LIN {X 0,Y 473.146,Z 970.34,A -85,B 0,C 180,E1 12740.095,E2 12740.095} C_VEL
LIN {X 0,Y 467.036,Z 990.213,A -85,B 0,C 180,E1 12738.717,E2 12738.717} C_VEL
LIN {X 0,Y 459.248,Z 1013.166,A -85,B 0,C 180,E1 12736.833,E2 12736.833} C_VEL
LIN {X 0,Y 452.835,Z 1030.812,A -85,B 0,C 180,E1 12735.136,E2 12735.136} C_VEL
LIN {X 0,Y 446.449,Z 1047.58,A -85,B 0,C 180,E1 12733.29,E2 12733.29} C_VEL
LIN {X 0,Y 438.433,Z 1067.669,A -85,B 0,C 180,E1 12730.711,E2 12730.711} C_VEL
LIN {X 0,Y 431.964,Z 1083.373,A -85,B 0,C 180,E1 12728.342,E2 12728.342} C_VEL
LIN {X 0,Y 426.155,Z 1097.416,A -85,B 0,C 180,E1 12725.914,E2 12725.914} C_VEL
LIN {X 0,Y 419.42,Z 1113.778,A -85,B 0,C 180,E1 12722.601,E2 12722.601} C_VEL
LIN {X 0,Y 414.613,Z 1125.727,A -85,B 0,C 180,E1 12719.751,E2 12719.751} C_VEL
LIN {X 0,Y 410.531,Z 1136.515,A -85,B 0,C 180,E1 12716.781,E2 12716.781} C_VEL
LIN {X 0,Y 406.512,Z 1147.962,A -85,B 0,C 180,E1 12713.022,E2 12713.022} C_VEL
LIN {X 0,Y 404.065,Z 1155.889,A -85,B 0,C 180,E1 12709.891,E2 12709.891} C_VEL
LIN {X 0,Y 402.255,Z 1162.846,A -85,B 0,C 180,E1 12706.61,E2 12706.61} C_VEL
LIN {X 0,Y 400.903,Z 1169.393,A -85,B 0,C 180,E1 12702.679,E2 12702.679} C_VEL
LIN {X 0,Y 400.333,Z 1173.356,A -85,B 0,C 180,E1 12699.488,E2 12699.488} C_VEL
LIN {X 0,Y 400.081,Z 1175.968,A -85,B 0,C 180,E1 12696.602,E2 12696.602} C_VEL
LIN {X 0,Y 399.979,Z 1177.638,A -85,B 0,C 180,E1 12693.743,E2 12693.743} C_VEL
LIN {X 0,Y 398.967,Z 1178.164,A -85,B 0,C 180,E1 12692.642,E2 12692.642} C_VEL
LIN {X 0,Y 392.498,Z 1178.722,A -85,B 0,C 180,E1 12689.533,E2 12689.533} C_VEL
LIN {X 0,Y 391.968,Z 1178.604,A -85,B 0,C 180,E1 12688.72,E2 12688.72} C_VEL
LIN {X 0,Y 391.987,Z 1177.784,A -85,B 0,C 180,E1 12685.85,E2 12685.85} C_VEL
LIN {X 0,Y 392.101,Z 1176.075,A -85,B 0,C 180,E1 12682.97,E2 12682.97} C_VEL
LIN {X 0,Y 392.411,Z 1173.254,A -85,B 0,C 180,E1 12679.874,E2 12679.874} C_VEL
LIN {X 0,Y 393.255,Z 1168.327,A -85,B 0,C 180,E1 12676.023,E2 12676.023} C_VEL
LIN {X 0,Y 394.664,Z 1162.136,A -85,B 0,C 180,E1 12672.454,E2 12672.454} C_VEL
LIN {X 0,Y 396.579,Z 1155.443,A -85,B 0,C 180,E1 12669.294,E2 12669.294} C_VEL
LIN {X 0,Y 399.73,Z 1146.131,A -85,B 0,C 180,E1 12665.624,E2 12665.624} C_VEL
LIN {X 0,Y 403.819,Z 1135.113,A -85,B 0,C 180,E1 12662.097,E2 12662.097} C_VEL
LIN {X 0,Y 408.079,Z 1124.561,A -85,B 0,C 180,E1 12659.197,E2 12659.197} C_VEL
LIN {X 0,Y 413.992,Z 1110.691,A -85,B 0,C 180,E1 12655.922,E2 12655.922} C_VEL
LIN {X 0,Y 420.293,Z 1095.933,A -85,B 0,C 180,E1 12652.995,E2 12652.995} C_VEL
LIN {X 0,Y 426.436,Z 1081.715,A -85,B 0,C 180,E1 12650.549,E2 12650.549} C_VEL
LIN {X 0,Y 434.19,Z 1063.573,A -85,B 0,C 180,E1 12647.862,E2 12647.862} C_VEL
LIN {X 0,Y 441.406,Z 1045.876,A -85,B 0,C 180,E1 12645.641,E2 12645.641} C_VEL
LIN {X 0,Y 447.609,Z 1030.103,A -85,B 0,C 180,E1 12643.912,E2 12643.912} C_VEL
LIN {X 0,Y 454.558,Z 1011.557,A -85,B 0,C 180,E1 12642.138,E2 12642.138} C_VEL
LIN {X 0,Y 462.542,Z 988.401,A -85,B 0,C 180,E1 12640.264,E2 12640.264} C_VEL
LIN {X 0,Y 468.329,Z 970.074,A -85,B 0,C 180,E1 12639.001,E2 12639.001} C_VEL
LIN {X 0,Y 473.769,Z 951.275,A -85,B 0,C 180,E1 12637.879,E2 12637.879} C_VEL
LIN {X 0,Y 479.972,Z 927.543,A -85,B 0,C 180,E1 12636.676,E2 12636.676} C_VEL
LIN {X 0,Y 485.302,Z 903.176,A -85,B 0,C 180,E1 12635.682,E2 12635.682} C_VEL
LIN {X 0,Y 489.311,Z 881.807,A -85,B 0,C 180,E1 12634.974,E2 12634.974} C_VEL
LIN {X 0,Y 492.754,Z 859.731,A -85,B 0,C 180,E1 12634.388,E2 12634.388} C_VEL
LIN {X 0,Y 495.9,Z 831.506,A -85,B 0,C 180,E1 12633.822,E2 12633.822} C_VEL
LIN {X 0,Y 501.269,Z 744.172,A -85,B 0,C 180,E1 12632.472,E2 12632.472} C_VEL
LIN {X 0,Y 515.214,Z 519.075,A -85,B 0,C 180,E1 12629.039,E2 12629.039} C_VEL
LIN {X 0,Y 515.608,Z 511.707,A -85,B 0,C 180,E1 12628.908,E2 12628.908} C_VEL
LIN {X 0,Y 507.102,Z 497.155,A -85,B 0,C 180,E1 12626.463,E2 12626.463} C_VEL
LIN {X 0,Y 498.411,Z 483.085,A -85,B 0,C 180,E1 12623.624,E2 12623.624} C_VEL
LIN {X 0,Y 491.406,Z 472.463,A -85,B 0,C 180,E1 12620.985,E2 12620.985} C_VEL
LIN {X 0,Y 485.728,Z 463.88,A -85,B 0,C 180,E1 12618.483,E2 12618.483} C_VEL
LIN {X 0,Y 479.648,Z 454.966,A -85,B 0,C 180,E1 12615.228,E2 12615.228} C_VEL
LIN {X 0,Y 475.792,Z 449.569,A -85,B 0,C 180,E1 12612.624,E2 12612.624} C_VEL
LIN {X 0,Y 472.697,Z 444.935,A -85,B 0,C 180,E1 12609.866,E2 12609.866} C_VEL
LIN {X 0,Y 469.6,Z 440.032,A -85,B 0,C 180,E1 12605.008,E2 12605.008} C_VEL
LIN {X 0,Y 469.247,Z 439.353,A -85,B 0,C 180,E1 12600.61,E2 12600.61} C_VEL
LIN {X 0,Y 471.413,Z 440.805,A -85,B 0,C 180,E1 12596.23,E2 12596.23} C_VEL
LIN {X 0,Y 476.457,Z 446.858,A -85,B 0,C 180,E1 12591.431,E2 12591.431} C_VEL
LIN {X 0,Y 481.036,Z 452.574,A -85,B 0,C 180,E1 12588.489,E2 12588.489} C_VEL
LIN {X 0,Y 485.576,Z 458.421,A -85,B 0,C 180,E1 12586.12,E2 12586.12} C_VEL
LIN {X 0,Y 489.604,Z 463.69,A -85,B 0,C 180,E1 12584.3,E2 12584.3} C_VEL
LIN {X 0,Y 494.319,Z 470.066,A -85,B 0,C 180,E1 12582.398,E2 12582.398} C_VEL
LIN {X 0,Y 500.346,Z 478.471,A -85,B 0,C 180,E1 12580.231,E2 12580.231} C_VEL
LIN {X 0,Y 508.251,Z 489.865,A -85,B 0,C 180,E1 12577.716,E2 12577.716} C_VEL
LIN {X 0,Y 517.057,Z 503.62,A -85,B 0,C 180,E1 12575.219,E2 12575.219} C_VEL
LIN {X 0,Y 518.568,Z 506.345,A -85,B 0,C 180,E1 12574.808,E2 12574.808} C_VEL
LIN {X 0,Y 504.377,Z 721.683,A -85,B 0,C 180,E1 12571.385,E2 12571.385} C_VEL
LIN {X 0,Y 497.461,Z 827.352,A -85,B 0,C 180,E1 12569.683,E2 12569.683} C_VEL
LIN {X 0,Y 494.393,Z 855.041,A -85,B 0,C 180,E1 12569.129,E2 12569.129} C_VEL
LIN {X 0,Y 490.441,Z 880.362,A -85,B 0,C 180,E1 12568.45,E2 12568.45} C_VEL
LIN {X 0,Y 486.512,Z 901.447,A -85,B 0,C 180,E1 12567.748,E2 12567.748} C_VEL
LIN {X 0,Y 482.08,Z 922.13,A -85,B 0,C 180,E1 12566.922,E2 12566.922} C_VEL
LIN {X 0,Y 476.116,Z 946.785,A -85,B 0,C 180,E1 12565.748,E2 12565.748} C_VEL
LIN {X 0,Y 469.403,Z 970.831,A -85,B 0,C 180,E1 12564.354,E2 12564.354} C_VEL
LIN {X 0,Y 463.52,Z 990.123,A -85,B 0,C 180,E1 12563.055,E2 12563.055} C_VEL
LIN {X 0,Y 457.46,Z 1008.652,A -85,B 0,C 180,E1 12561.629,E2 12561.629} C_VEL
LIN {X 0,Y 450.307,Z 1029.319,A -85,B 0,C 180,E1 12559.802,E2 12559.802} C_VEL
LIN {X 0,Y 442.12,Z 1051.496,A -85,B 0,C 180,E1 12557.499,E2 12557.499} C_VEL
LIN {X 0,Y 435.558,Z 1068.547,A -85,B 0,C 180,E1 12555.453,E2 12555.453} C_VEL
LIN {X 0,Y 429.309,Z 1084.464,A -85,B 0,C 180,E1 12553.287,E2 12553.287} C_VEL
LIN {X 0,Y 422.177,Z 1102.656,A -85,B 0,C 180,E1 12550.461,E2 12550.461} C_VEL
LIN {X 0,Y 415.361,Z 1119.695,A -85,B 0,C 180,E1 12547.346,E2 12547.346} C_VEL
LIN {X 0,Y 410.527,Z 1132.16,A -85,B 0,C 180,E1 12544.745,E2 12544.745} C_VEL
LIN {X 0,Y 406.154,Z 1143.963,A -85,B 0,C 180,E1 12541.957,E2 12541.957} C_VEL
LIN {X 0,Y 401.616,Z 1157.152,A -85,B 0,C 180,E1 12538.393,E2 12538.393} C_VEL
LIN {X 0,Y 398.108,Z 1168.263,A -85,B 0,C 180,E1 12534.798,E2 12534.798} C_VEL
LIN {X 0,Y 395.81,Z 1176.642,A -85,B 0,C 180,E1 12531.642,E2 12531.642} C_VEL
LIN {X 0,Y 394.214,Z 1183.474,A -85,B 0,C 180,E1 12528.637,E2 12528.637} C_VEL
LIN {X 0,Y 393.104,Z 1189.495,A -85,B 0,C 180,E1 12525.49,E2 12525.49} C_VEL
LIN {X 0,Y 392.374,Z 1194.808,A -85,B 0,C 180,E1 12522.061,E2 12522.061} C_VEL
LIN {X 0,Y 392.03,Z 1199.164,A -85,B 0,C 180,E1 12518.211,E2 12518.211} C_VEL
LIN {X 0,Y 391.945,Z 1201.596,A -85,B 0,C 180,E1 12514.829,E2 12514.829} C_VEL
LIN {X 0,Y 391.936,Z 1202.702,A -85,B 0,C 180,E1 12511.9,E2 12511.9} C_VEL
LIN {X 0,Y 391.937,Z 1202.845,A -85,B 0,C 180,E1 12508.976,E2 12508.976} C_VEL
LIN {X 0,Y 391.938,Z 1202.024,A -85,B 0,C 180,E1 12506.05,E2 12506.05} C_VEL
LIN {X 0,Y 391.978,Z 1200.238,A -85,B 0,C 180,E1 12503.114,E2 12503.114} C_VEL
LIN {X 0,Y 392.133,Z 1197.477,A -85,B 0,C 180,E1 12500.163,E2 12500.163} C_VEL
LIN {X 0,Y 392.488,Z 1193.725,A -85,B 0,C 180,E1 12497.195,E2 12497.195} C_VEL
LIN {X 0,Y 393.191,Z 1188.961,A -85,B 0,C 180,E1 12494.21,E2 12494.21} C_VEL
LIN {X 0,Y 394.28,Z 1183.151,A -85,B 0,C 180,E1 12491.212,E2 12491.212} C_VEL
LIN {X 0,Y 395.905,Z 1176.264,A -85,B 0,C 180,E1 12488.207,E2 12488.207} C_VEL
LIN {X 0,Y 398.362,Z 1167.411,A -85,B 0,C 180,E1 12484.901,E2 12484.901} C_VEL
LIN {X 0,Y 402.48,Z 1154.483,A -85,B 0,C 180,E1 12480.861,E2 12480.861} C_VEL
LIN {X 0,Y 406.36,Z 1143.356,A -85,B 0,C 180,E1 12477.894,E2 12477.894} C_VEL
LIN {X 0,Y 410.781,Z 1131.482,A -85,B 0,C 180,E1 12475.109,E2 12475.109} C_VEL
LIN {X 0,Y 416.541,Z 1116.774,A -85,B 0,C 180,E1 12472.083,E2 12472.083} C_VEL
LIN {X 0,Y 423.481,Z 1099.133,A -85,B 0,C 180,E1 12468.975,E2 12468.975} C_VEL
LIN {X 0,Y 429.75,Z 1083.261,A -85,B 0,C 180,E1 12466.546,E2 12466.546} C_VEL
LIN {X 0,Y 436.179,Z 1066.874,A -85,B 0,C 180,E1 12464.339,E2 12464.339} C_VEL
LIN {X 0,Y 444.324,Z 1045.603,A -85,B 0,C 180,E1 12461.853,E2 12461.853} C_VEL
LIN {X 0,Y 451.719,Z 1025.122,A -85,B 0,C 180,E1 12459.818,E2 12459.818} C_VEL
LIN {X 0,Y 458.1,Z 1006.573,A -85,B 0,C 180,E1 12458.209,E2 12458.209} C_VEL
LIN {X 0,Y 464.819,Z 985.852,A -85,B 0,C 180,E1 12456.643,E2 12456.643} C_VEL
LIN {X 0,Y 472.394,Z 960.109,A -85,B 0,C 180,E1 12455.002,E2 12455.002} C_VEL
LIN {X 0,Y 478.021,Z 938.783,A -85,B 0,C 180,E1 12453.859,E2 12453.859} C_VEL
LIN {X 0,Y 482.942,Z 917.99,A -85,B 0,C 180,E1 12452.908,E2 12452.908} C_VEL
LIN {X 0,Y 488.168,Z 892.954,A -85,B 0,C 180,E1 12451.953,E2 12451.953} C_VEL
LIN {X 0,Y 492.624,Z 866.372,A -85,B 0,C 180,E1 12451.161,E2 12451.161} C_VEL
LIN {X 0,Y 495.65,Z 843.976,A -85,B 0,C 180,E1 12450.64,E2 12450.64} C_VEL
LIN {X 0,Y 497.907,Z 820.907,A -85,B 0,C 180,E1 12450.212,E2 12450.212} C_VEL
LIN {X 0,Y 512.049,Z 602.752,A -85,B 0,C 180,E1 12446.728,E2 12446.728} C_VEL
LIN {X 0,Y 518.415,Z 505.981,A -85,B 0,C 180,E1 12445.175,E2 12445.175} C_VEL
LIN {X 0,Y 510.173,Z 492.964,A -85,B 0,C 180,E1 12442.895,E2 12442.895} C_VEL
LIN {X 0,Y 502.413,Z 481.412,A -85,B 0,C 180,E1 12440.504,E2 12440.504} C_VEL
LIN {X 0,Y 494.907,Z 470.885,A -85,B 0,C 180,E1 12437.884,E2 12437.884} C_VEL
LIN {X 0,Y 488.282,Z 461.837,A -85,B 0,C 180,E1 12435.196,E2 12435.196} C_VEL
LIN {X 0,Y 483.762,Z 456.181,A -85,B 0,C 180,E1 12433.081,E2 12433.081} C_VEL
LIN {X 0,Y 479.837,Z 451.127,A -85,B 0,C 180,E1 12430.931,E2 12430.931} C_VEL
LIN {X 0,Y 475.767,Z 446.066,A -85,B 0,C 180,E1 12428.216,E2 12428.216} C_VEL
LIN {X 0,Y 471.079,Z 440.513,A -85,B 0,C 180,E1 12423.651,E2 12423.651} C_VEL
LIN {X 0,Y 468.928,Z 439.119,A -85,B 0,C 180,E1 12419.145,E2 12419.145} C_VEL
LIN {X 0,Y 469.43,Z 439.93,A -85,B 0,C 180,E1 12414.622,E2 12414.622} C_VEL
LIN {X 0,Y 473.229,Z 445.796,A -85,B 0,C 180,E1 12409.284,E2 12409.284} C_VEL
LIN {X 0,Y 476.763,Z 451.073,A -85,B 0,C 180,E1 12406.415,E2 12406.415} C_VEL
LIN {X 0,Y 480.383,Z 456.255,A -85,B 0,C 180,E1 12404.115,E2 12404.115} C_VEL
LIN {X 0,Y 486.229,Z 464.697,A -85,B 0,C 180,E1 12401.102,E2 12401.102} C_VEL
LIN {X 0,Y 492.378,Z 473.967,A -85,B 0,C 180,E1 12398.466,E2 12398.466} C_VEL
LIN {X 0,Y 500.014,Z 485.785,A -85,B 0,C 180,E1 12395.673,E2 12395.673} C_VEL
LIN {X 0,Y 508.042,Z 498.9,A -85,B 0,C 180,E1 12393.116,E2 12393.116} C_VEL
LIN {X 0,Y 515.57,Z 511.771,A -85,B 0,C 180,E1 12390.975,E2 12390.975} C_VEL
LIN {X 0,Y 501.344,Z 741.185,A -85,B 0,C 180,E1 12387.476,E2 12387.476} C_VEL
LIN {X 0,Y 495.804,Z 831.47,A -85,B 0,C 180,E1 12386.082,E2 12386.082} C_VEL
LIN {X 0,Y 492.648,Z 859.813,A -85,B 0,C 180,E1 12385.512,E2 12385.512} C_VEL
LIN {X 0,Y 489.23,Z 881.718,A -85,B 0,C 180,E1 12384.932,E2 12384.932} C_VEL
LIN {X 0,Y 485.22,Z 903.138,A -85,B 0,C 180,E1 12384.222,E2 12384.222} C_VEL
LIN {X 0,Y 479.632,Z 928.52,A -85,B 0,C 180,E1 12383.18,E2 12383.18} C_VEL
LIN {X 0,Y 473.724,Z 951.145,A -85,B 0,C 180,E1 12382.031,E2 12382.031} C_VEL
LIN {X 0,Y 468.292,Z 969.947,A -85,B 0,C 180,E1 12380.908,E2 12380.908} C_VEL
LIN {X 0,Y 462.254,Z 989.07,A -85,B 0,C 180,E1 12379.587,E2 12379.587} C_VEL
LIN {X 0,Y 454.226,Z 1012.249,A -85,B 0,C 180,E1 12377.7,E2 12377.7} C_VEL
LIN {X 0,Y 447.538,Z 1030.126,A -85,B 0,C 180,E1 12375.985,E2 12375.985} C_VEL
LIN {X 0,Y 441.108,Z 1046.484,A -85,B 0,C 180,E1 12374.189,E2 12374.189} C_VEL
LIN {X 0,Y 433.453,Z 1065.279,A -85,B 0,C 180,E1 12371.81,E2 12371.81} C_VEL
LIN {X 0,Y 426.144,Z 1082.288,A -85,B 0,C 180,E1 12369.258,E2 12369.258} C_VEL
LIN {X 0,Y 420.336,Z 1095.748,A -85,B 0,C 180,E1 12366.939,E2 12366.939} C_VEL
LIN {X 0,Y 414.13,Z 1110.273,A -85,B 0,C 180,E1 12364.066,E2 12364.066} C_VEL
LIN {X 0,Y 408.209,Z 1124.219,A -85,B 0,C 180,E1 12360.793,E2 12360.793} C_VEL
LIN {X 0,Y 403.927,Z 1134.806,A -85,B 0,C 180,E1 12357.895,E2 12357.895} C_VEL
LIN {X 0,Y 399.964,Z 1145.412,A -85,B 0,C 180,E1 12354.519,E2 12354.519} C_VEL
LIN {X 0,Y 396.67,Z 1155.135,A -85,B 0,C 180,E1 12350.741,E2 12350.741} C_VEL
LIN {X 0,Y 394.71,Z 1161.947,A -85,B 0,C 180,E1 12347.545,E2 12347.545} C_VEL
LIN {X 0,Y 393.326,Z 1167.924,A -85,B 0,C 180,E1 12344.126,E2 12344.126} C_VEL
LIN {X 0,Y 392.422,Z 1173.153,A -85,B 0,C 180,E1 12340.126,E2 12340.126} C_VEL
LIN {X 0,Y 392.106,Z 1176.002,A -85,B 0,C 180,E1 12337.031,E2 12337.031} C_VEL
LIN {X 0,Y 391.991,Z 1177.764,A -85,B 0,C 180,E1 12334.096,E2 12334.096} C_VEL
LIN {X 0,Y 391.967,Z 1178.606,A -85,B 0,C 180,E1 12331.17,E2 12331.17} C_VEL
LIN {X 0,Y 391.968,Z 1178.604,A -85,B 0,C 180,E1 12328.72,E2 12328.72} C_VEL
LIN {X 0,Y 390.977,Z 1178.483,A -85,B 0,C 180,E1 12327.594,E2 12327.594} C_VEL
LIN {X 0,Y 384.565,Z 1177.435,A -85,B 0,C 180,E1 12324.42,E2 12324.42} C_VEL
LIN {X 0,Y 384.077,Z 1176.88,A -85,B 0,C 180,E1 12323.594,E2 12323.594} C_VEL
LIN {X 0,Y 384.354,Z 1174.24,A -85,B 0,C 180,E1 12320.39,E2 12320.39} C_VEL
LIN {X 0,Y 384.926,Z 1170.624,A -85,B 0,C 180,E1 12317.245,E2 12317.245} C_VEL
LIN {X 0,Y 386.013,Z 1165.662,A -85,B 0,C 180,E1 12313.91,E2 12313.91} C_VEL
LIN {X 0,Y 388.229,Z 1157.829,A -85,B 0,C 180,E1 12309.812,E2 12309.812} C_VEL
LIN {X 0,Y 390.887,Z 1149.923,A -85,B 0,C 180,E1 12306.482,E2 12306.482} C_VEL
LIN {X 0,Y 394.232,Z 1141.088,A -85,B 0,C 180,E1 12303.326,E2 12303.326} C_VEL
LIN {X 0,Y 399.571,Z 1128.179,A -85,B 0,C 180,E1 12299.471,E2 12299.471} C_VEL
LIN {X 0,Y 404.619,Z 1116.589,A -85,B 0,C 180,E1 12296.56,E2 12296.56} C_VEL
LIN {X 0,Y 410.183,Z 1104.168,A -85,B 0,C 180,E1 12293.85,E2 12293.85} C_VEL
LIN {X 0,Y 417.912,Z 1086.977,A -85,B 0,C 180,E1 12290.653,E2 12290.653} C_VEL
LIN {X 0,Y 424.722,Z 1071.574,A -85,B 0,C 180,E1 12288.223,E2 12288.223} C_VEL
LIN {X 0,Y 431.557,Z 1055.813,A -85,B 0,C 180,E1 12286.06,E2 12286.06} C_VEL
LIN {X 0,Y 440.337,Z 1034.648,A -85,B 0,C 180,E1 12283.585,E2 12283.585} C_VEL
LIN {X 0,Y 447.324,Z 1016.69,A -85,B 0,C 180,E1 12281.802,E2 12281.802} C_VEL
LIN {X 0,Y 453.924,Z 998.684,A -85,B 0,C 180,E1 12280.249,E2 12280.249} C_VEL
LIN {X 0,Y 461.658,Z 975.885,A -85,B 0,C 180,E1 12278.569,E2 12278.569} C_VEL
LIN {X 0,Y 468.311,Z 953.784,A -85,B 0,C 180,E1 12277.215,E2 12277.215} C_VEL
LIN {X 0,Y 473.763,Z 933.72,A -85,B 0,C 180,E1 12276.171,E2 12276.171} C_VEL
LIN {X 0,Y 479.651,Z 909.21,A -85,B 0,C 180,E1 12275.106,E2 12275.106} C_VEL
LIN {X 0,Y 484.517,Z 884.316,A -85,B 0,C 180,E1 12274.254,E2 12274.254} C_VEL
LIN {X 0,Y 487.846,Z 863.962,A -85,B 0,C 180,E1 12273.697,E2 12273.697} C_VEL
LIN {X 0,Y 490.821,Z 840.782,A -85,B 0,C 180,E1 12273.194,E2 12273.194} C_VEL
LIN {X 0,Y 493.481,Z 805.983,A -85,B 0,C 180,E1 12272.62,E2 12272.62} C_VEL
LIN {X 0,Y 507.621,Z 579.641,A -85,B 0,C 180,E1 12269.16,E2 12269.16} C_VEL
LIN {X 0,Y 511.778,Z 516.311,A -85,B 0,C 180,E1 12268.188,E2 12268.188} C_VEL
LIN {X 0,Y 503.439,Z 501.906,A -85,B 0,C 180,E1 12265.688,E2 12265.688} C_VEL
LIN {X 0,Y 495.488,Z 489.034,A -85,B 0,C 180,E1 12262.985,E2 12262.985} C_VEL
LIN {X 0,Y 489.537,Z 479.735,A -85,B 0,C 180,E1 12260.662,E2 12260.662} C_VEL
LIN {X 0,Y 483.92,Z 471.102,A -85,B 0,C 180,E1 12258.118,E2 12258.118} C_VEL
LIN {X 0,Y 478.097,Z 462.45,A -85,B 0,C 180,E1 12254.907,E2 12254.907} C_VEL
LIN {X 0,Y 474.51,Z 457.281,A -85,B 0,C 180,E1 12252.412,E2 12252.412} C_VEL
LIN {X 0,Y 471.613,Z 452.818,A -85,B 0,C 180,E1 12249.765,E2 12249.765} C_VEL
LIN {X 0,Y 468.583,Z 447.936,A -85,B 0,C 180,E1 12244.896,E2 12244.896} C_VEL
LIN {X 0,Y 468.298,Z 447.304,A -85,B 0,C 180,E1 12240.489,E2 12240.489} C_VEL
LIN {X 0,Y 470.427,Z 448.822,A -85,B 0,C 180,E1 12236.222,E2 12236.222} C_VEL
LIN {X 0,Y 475.224,Z 454.666,A -85,B 0,C 180,E1 12231.591,E2 12231.591} C_VEL
LIN {X 0,Y 479.632,Z 460.264,A -85,B 0,C 180,E1 12228.699,E2 12228.699} C_VEL
LIN {X 0,Y 483.985,Z 465.951,A -85,B 0,C 180,E1 12226.378,E2 12226.378} C_VEL
LIN {X 0,Y 488.07,Z 471.415,A -85,B 0,C 180,E1 12224.493,E2 12224.493} C_VEL
LIN {X 0,Y 494.049,Z 479.506,A -85,B 0,C 180,E1 12222.084,E2 12222.084} C_VEL
LIN {X 0,Y 502.08,Z 491.222,A -85,B 0,C 180,E1 12219.268,E2 12219.268} C_VEL
LIN {X 0,Y 510.053,Z 503.319,A -85,B 0,C 180,E1 12216.825,E2 12216.825} C_VEL
LIN {X 0,Y 514.618,Z 510.925,A -85,B 0,C 180,E1 12215.531,E2 12215.531} C_VEL
LIN {X 0,Y 499.932,Z 727.913,A -85,B 0,C 180,E1 12212.078,E2 12212.078} C_VEL
LIN {X 0,Y 493.21,Z 827.545,A -85,B 0,C 180,E1 12210.468,E2 12210.468} C_VEL
LIN {X 0,Y 490.042,Z 855.381,A -85,B 0,C 180,E1 12209.911,E2 12209.911} C_VEL
LIN {X 0,Y 486.039,Z 880.426,A -85,B 0,C 180,E1 12209.241,E2 12209.241} C_VEL
LIN {X 0,Y 482.041,Z 901.406,A -85,B 0,C 180,E1 12208.543,E2 12208.543} C_VEL
LIN {X 0,Y 477.377,Z 922.606,A -85,B 0,C 180,E1 12207.698,E2 12207.698} C_VEL
LIN {X 0,Y 471.179,Z 947.492,A -85,B 0,C 180,E1 12206.509,E2 12206.509} C_VEL
LIN {X 0,Y 464.346,Z 971.239,A -85,B 0,C 180,E1 12205.125,E2 12205.125} C_VEL
LIN {X 0,Y 458.301,Z 990.477,A -85,B 0,C 180,E1 12203.826,E2 12203.826} C_VEL
LIN {X 0,Y 451.739,Z 1009.928,A -85,B 0,C 180,E1 12202.316,E2 12202.316} C_VEL
LIN {X 0,Y 443.502,Z 1032.867,A -85,B 0,C 180,E1 12200.244,E2 12200.244} C_VEL
LIN {X 0,Y 435.783,Z 1052.875,A -85,B 0,C 180,E1 12198.111,E2 12198.111} C_VEL
LIN {X 0,Y 429.074,Z 1069.692,A -85,B 0,C 180,E1 12196.059,E2 12196.059} C_VEL
LIN {X 0,Y 422.095,Z 1086.865,A -85,B 0,C 180,E1 12193.671,E2 12193.671} C_VEL
LIN {X 0,Y 414.059,Z 1106.318,A -85,B 0,C 180,E1 12190.51,E2 12190.51} C_VEL
LIN {X 0,Y 408.366,Z 1120.097,A -85,B 0,C 180,E1 12187.92,E2 12187.92} C_VEL
LIN {X 0,Y 403.343,Z 1132.503,A -85,B 0,C 180,E1 12185.282,E2 12185.282} C_VEL
LIN {X 0,Y 398.528,Z 1144.951,A -85,B 0,C 180,E1 12182.272,E2 12182.272} C_VEL
LIN {X 0,Y 393.36,Z 1159.25,A -85,B 0,C 180,E1 12178.215,E2 12178.215} C_VEL
LIN {X 0,Y 390.255,Z 1168.818,A -85,B 0,C 180,E1 12175.008,E2 12175.008} C_VEL
LIN {X 0,Y 387.956,Z 1176.833,A -85,B 0,C 180,E1 12171.899,E2 12171.899} C_VEL
LIN {X 0,Y 386.243,Z 1183.831,A -85,B 0,C 180,E1 12168.723,E2 12168.723} C_VEL
LIN {X 0,Y 384.982,Z 1190.554,A -85,B 0,C 180,E1 12165.053,E2 12165.053} C_VEL
LIN {X 0,Y 384.245,Z 1196.047,A -85,B 0,C 180,E1 12161.102,E2 12161.102} C_VEL
LIN {X 0,Y 384.013,Z 1199.39,A -85,B 0,C 180,E1 12157.781,E2 12157.781} C_VEL
LIN {X 0,Y 383.947,Z 1201.418,A -85,B 0,C 180,E1 12154.78,E2 12154.78} C_VEL
LIN {X 0,Y 383.94,Z 1202.479,A -85,B 0,C 180,E1 12151.791,E2 12151.791} C_VEL
LIN {X 0,Y 383.941,Z 1202.598,A -85,B 0,C 180,E1 12148.955,E2 12148.955} C_VEL
LIN {X 0,Y 383.941,Z 1201.744,A -85,B 0,C 180,E1 12145.904,E2 12145.904} C_VEL
LIN {X 0,Y 383.985,Z 1199.984,A -85,B 0,C 180,E1 12142.97,E2 12142.97} C_VEL
LIN {X 0,Y 384.15,Z 1197.218,A -85,B 0,C 180,E1 12139.957,E2 12139.957} C_VEL
LIN {X 0,Y 384.532,Z 1193.461,A -85,B 0,C 180,E1 12136.925,E2 12136.925} C_VEL
LIN {X 0,Y 385.285,Z 1188.69,A -85,B 0,C 180,E1 12133.878,E2 12133.878} C_VEL
LIN {X 0,Y 386.466,Z 1182.832,A -85,B 0,C 180,E1 12130.796,E2 12130.796} C_VEL
LIN {X 0,Y 388.295,Z 1175.588,A -85,B 0,C 180,E1 12127.587,E2 12127.587} C_VEL
LIN {X 0,Y 391.391,Z 1165.306,A -85,B 0,C 180,E1 12123.729,E2 12123.729} C_VEL
LIN {X 0,Y 395.32,Z 1153.646,A -85,B 0,C 180,E1 12120.114,E2 12120.114} C_VEL
LIN {X 0,Y 399.223,Z 1143.046,A -85,B 0,C 180,E1 12117.249,E2 12117.249} C_VEL
LIN {X 0,Y 403.877,Z 1131.166,A -85,B 0,C 180,E1 12114.423,E2 12114.423} C_VEL
LIN {X 0,Y 410.013,Z 1116.152,A -85,B 0,C 180,E1 12111.296,E2 12111.296} C_VEL
LIN {X 0,Y 417.155,Z 1098.708,A -85,B 0,C 180,E1 12108.198,E2 12108.198} C_VEL
LIN {X 0,Y 423.417,Z 1083.48,A -85,B 0,C 180,E1 12105.843,E2 12105.843} C_VEL
LIN {X 0,Y 429.903,Z 1067.544,A -85,B 0,C 180,E1 12103.67,E2 12103.67} C_VEL
LIN {X 0,Y 438.079,Z 1047.052,A -85,B 0,C 180,E1 12101.231,E2 12101.231} C_VEL
LIN {X 0,Y 445.916,Z 1026.06,A -85,B 0,C 180,E1 12099.119,E2 12099.119} C_VEL
LIN {X 0,Y 452.471,Z 1007.621,A -85,B 0,C 180,E1 12097.502,E2 12097.502} C_VEL
LIN {X 0,Y 459.066,Z 987.931,A -85,B 0,C 180,E1 12095.997,E2 12095.997} C_VEL
LIN {X 0,Y 466.583,Z 963.622,A -85,B 0,C 180,E1 12094.406,E2 12094.406} C_VEL
LIN {X 0,Y 472.895,Z 940.444,A -85,B 0,C 180,E1 12093.144,E2 12093.144} C_VEL
LIN {X 0,Y 477.928,Z 919.88,A -85,B 0,C 180,E1 12092.193,E2 12092.193} C_VEL
LIN {X 0,Y 482.491,Z 898.865,A -85,B 0,C 180,E1 12091.373,E2 12091.373} C_VEL
LIN {X 0,Y 487.31,Z 872.956,A -85,B 0,C 180,E1 12090.542,E2 12090.542} C_VEL
LIN {X 0,Y 491.092,Z 846.31,A -85,B 0,C 180,E1 12089.899,E2 12089.899} C_VEL
LIN {X 0,Y 493.443,Z 823.735,A -85,B 0,C 180,E1 12089.472,E2 12089.472} C_VEL
LIN {X 0,Y 507.6,Z 611.937,A -85,B 0,C 180,E1 12086.081,E2 12086.081} C_VEL
LIN {X 0,Y 514.463,Z 510.576,A -85,B 0,C 180,E1 12084.455,E2 12084.455} C_VEL
LIN {X 0,Y 506.12,Z 497.341,A -85,B 0,C 180,E1 12082.047,E2 12082.047} C_VEL
LIN {X 0,Y 498.62,Z 486.304,A -85,B 0,C 180,E1 12079.627,E2 12079.627} C_VEL
LIN {X 0,Y 492.432,Z 477.471,A -85,B 0,C 180,E1 12077.367,E2 12077.367} C_VEL
LIN {X 0,Y 486.506,Z 469.232,A -85,B 0,C 180,E1 12074.887,E2 12074.887} C_VEL
LIN {X 0,Y 482.311,Z 463.859,A -85,B 0,C 180,E1 12072.877,E2 12072.877} C_VEL
LIN {X 0,Y 478.452,Z 458.822,A -85,B 0,C 180,E1 12070.719,E2 12070.719} C_VEL
LIN {X 0,Y 474.459,Z 453.814,A -85,B 0,C 180,E1 12067.995,E2 12067.995} C_VEL
LIN {X 0,Y 470.007,Z 448.405,A -85,B 0,C 180,E1 12063.537,E2 12063.537} C_VEL
LIN {X 0,Y 467.932,Z 447.055,A -85,B 0,C 180,E1 12059.02,E2 12059.02} C_VEL
LIN {X 0,Y 468.458,Z 447.885,A -85,B 0,C 180,E1 12054.611,E2 12054.611} C_VEL
LIN {X 0,Y 472.068,Z 453.611,A -85,B 0,C 180,E1 12049.443,E2 12049.443} C_VEL
LIN {X 0,Y 475.454,Z 458.775,A -85,B 0,C 180,E1 12046.624,E2 12046.624} C_VEL
LIN {X 0,Y 479.008,Z 463.98,A -85,B 0,C 180,E1 12044.317,E2 12044.317} C_VEL
LIN {X 0,Y 484.584,Z 472.179,A -85,B 0,C 180,E1 12041.379,E2 12041.379} C_VEL
LIN {X 0,Y 490.556,Z 481.355,A -85,B 0,C 180,E1 12038.758,E2 12038.758} C_VEL
LIN {X 0,Y 497.989,Z 493.096,A -85,B 0,C 180,E1 12035.978,E2 12035.978} C_VEL
LIN {X 0,Y 505.725,Z 505.95,A -85,B 0,C 180,E1 12033.459,E2 12033.459} C_VEL
LIN {X 0,Y 511.681,Z 516.381,A -85,B 0,C 180,E1 12031.707,E2 12031.707} C_VEL
LIN {X 0,Y 497.135,Z 744.161,A -85,B 0,C 180,E1 12028.227,E2 12028.227} C_VEL
LIN {X 0,Y 491.597,Z 831.501,A -85,B 0,C 180,E1 12026.875,E2 12026.875} C_VEL
LIN {X 0,Y 488.34,Z 859.985,A -85,B 0,C 180,E1 12026.302,E2 12026.302} C_VEL
LIN {X 0,Y 484.829,Z 881.929,A -85,B 0,C 180,E1 12025.723,E2 12025.723} C_VEL
LIN {X 0,Y 480.786,Z 903.029,A -85,B 0,C 180,E1 12025.024,E2 12025.024} C_VEL
LIN {X 0,Y 475.178,Z 927.998,A -85,B 0,C 180,E1 12024.006,E2 12024.006} C_VEL
LIN {X 0,Y 468.828,Z 951.681,A -85,B 0,C 180,E1 12022.804,E2 12022.804} C_VEL
LIN {X 0,Y 462.981,Z 971.325,A -85,B 0,C 180,E1 12021.624,E2 12021.624} C_VEL
LIN {X 0,Y 455.749,Z 993.501,A -85,B 0,C 180,E1 12020.066,E2 12020.066} C_VEL
LIN {X 0,Y 448.043,Z 1014.611,A -85,B 0,C 180,E1 12018.287,E2 12018.287} C_VEL
LIN {X 0,Y 441.491,Z 1031.561,A -85,B 0,C 180,E1 12016.635,E2 12016.635} C_VEL
LIN {X 0,Y 434.618,Z 1048.472,A -85,B 0,C 180,E1 12014.748,E2 12014.748} C_VEL
LIN {X 0,Y 426.078,Z 1068.432,A -85,B 0,C 180,E1 12012.135,E2 12012.135} C_VEL
LIN {X 0,Y 419.544,Z 1083.181,A -85,B 0,C 180,E1 12009.874,E2 12009.874} C_VEL
LIN {X 0,Y 413.533,Z 1096.593,A -85,B 0,C 180,E1 12007.526,E2 12007.526} C_VEL
LIN {X 0,Y 406.735,Z 1111.895,A -85,B 0,C 180,E1 12004.431,E2 12004.431} C_VEL
LIN {X 0,Y 400.887,Z 1125.061,A -85,B 0,C 180,E1 12001.251,E2 12001.251} C_VEL
LIN {X 0,Y 396.439,Z 1135.585,A -85,B 0,C 180,E1 11998.305,E2 11998.305} C_VEL
LIN {X 0,Y 392.163,Z 1146.554,A -85,B 0,C 180,E1 11994.718,E2 11994.718} C_VEL
LIN {X 0,Y 388.896,Z 1155.689,A -85,B 0,C 180,E1 11991.042,E2 11991.042} C_VEL
LIN {X 0,Y 386.912,Z 1162.21,A -85,B 0,C 180,E1 11987.91,E2 11987.91} C_VEL
LIN {X 0,Y 385.435,Z 1168.184,A -85,B 0,C 180,E1 11984.421,E2 11984.421} C_VEL
LIN {X 0,Y 384.459,Z 1173.406,A -85,B 0,C 180,E1 11980.338,E2 11980.338} C_VEL
LIN {X 0,Y 384.123,Z 1176.252,A -85,B 0,C 180,E1 11977.178,E2 11977.178} C_VEL
LIN {X 0,Y 383.997,Z 1178.012,A -85,B 0,C 180,E1 11974.181,E2 11974.181} C_VEL
LIN {X 0,Y 383.97,Z 1178.853,A -85,B 0,C 180,E1 11971.194,E2 11971.194} C_VEL
LIN {X 0,Y 383.973,Z 1178.76,A -85,B 0,C 180,E1 11968.06,E2 11968.06} C_VEL
LIN {X 0,Y 384.042,Z 1177.404,A -85,B 0,C 180,E1 11964.322,E2 11964.322} C_VEL
LIN {X 0,Y 384.077,Z 1176.88,A -85,B 0,C 180,E1 11963.594,E2 11963.594} C_VEL
LIN {X 0,Y 383.168,Z 1176.104,A -85,B 0,C 180,E1 11962.449,E2 11962.449} C_VEL
LIN {X 0,Y 377.074,Z 1173.598,A -85,B 0,C 180,E1 11959.217,E2 11959.217} C_VEL
LIN {X 0,Y 376.688,Z 1172.681,A -85,B 0,C 180,E1 11958.382,E2 11958.382} C_VEL
LIN {X 0,Y 377.737,Z 1167.623,A -85,B 0,C 180,E1 11954.651,E2 11954.651} C_VEL
LIN {X 0,Y 379.256,Z 1162.076,A -85,B 0,C 180,E1 11951.398,E2 11951.398} C_VEL
LIN {X 0,Y 381.575,Z 1155.034,A -85,B 0,C 180,E1 11947.994,E2 11947.994} C_VEL
LIN {X 0,Y 385.602,Z 1144.463,A -85,B 0,C 180,E1 11943.845,E2 11943.845} C_VEL
LIN {X 0,Y 389.715,Z 1134.67,A -85,B 0,C 180,E1 11940.657,E2 11940.657} C_VEL
LIN {X 0,Y 394.794,Z 1123.369,A -85,B 0,C 180,E1 11937.5,E2 11937.5} C_VEL
LIN {X 0,Y 401.648,Z 1108.499,A -85,B 0,C 180,E1 11934.006,E2 11934.006} C_VEL
LIN {X 0,Y 407.588,Z 1095.783,A -85,B 0,C 180,E1 11931.457,E2 11931.457} C_VEL
LIN {X 0,Y 413.859,Z 1082.332,A -85,B 0,C 180,E1 11929.101,E2 11929.101} C_VEL
LIN {X 0,Y 422.137,Z 1064.287,A -85,B 0,C 180,E1 11926.373,E2 11926.373} C_VEL
LIN {X 0,Y 430.014,Z 1046.189,A -85,B 0,C 180,E1 11924.07,E2 11924.07} C_VEL
LIN {X 0,Y 436.947,Z 1029.634,A -85,B 0,C 180,E1 11922.246,E2 11922.246} C_VEL
LIN {X 0,Y 445.071,Z 1009.189,A -85,B 0,C 180,E1 11920.297,E2 11920.297} C_VEL
LIN {X 0,Y 452.793,Z 987.682,A -85,B 0,C 180,E1 11918.582,E2 11918.582} C_VEL
LIN {X 0,Y 458.929,Z 969.249,A -85,B 0,C 180,E1 11917.323,E2 11917.323} C_VEL
LIN {X 0,Y 464.672,Z 950.331,A -85,B 0,C 180,E1 11916.204,E2 11916.204} C_VEL
LIN {X 0,Y 471.196,Z 926.362,A -85,B 0,C 180,E1 11915.007,E2 11915.007} C_VEL
LIN {X 0,Y 476.643,Z 902.468,A -85,B 0,C 180,E1 11914.044,E2 11914.044} C_VEL
LIN {X 0,Y 480.835,Z 880.987,A -85,B 0,C 180,E1 11913.341,E2 11913.341} C_VEL
LIN {X 0,Y 484.925,Z 855.601,A -85,B 0,C 180,E1 11912.686,E2 11912.686} C_VEL
LIN {X 0,Y 487.765,Z 829.425,A -85,B 0,C 180,E1 11912.186,E2 11912.186} C_VEL
LIN {X 0,Y 502.364,Z 604.465,A -85,B 0,C 180,E1 11908.73,E2 11908.73} C_VEL
LIN {X 0,Y 507.943,Z 520.678,A -85,B 0,C 180,E1 11907.428,E2 11907.428} C_VEL
LIN {X 0,Y 500.018,Z 507.075,A -85,B 0,C 180,E1 11904.957,E2 11904.957} C_VEL
LIN {X 0,Y 493.304,Z 495.966,A -85,B 0,C 180,E1 11902.588,E2 11902.588} C_VEL
LIN {X 0,Y 487.551,Z 486.801,A -85,B 0,C 180,E1 11900.279,E2 11900.279} C_VEL
LIN {X 0,Y 482.013,Z 478.17,A -85,B 0,C 180,E1 11897.692,E2 11897.692} C_VEL
LIN {X 0,Y 476.656,Z 470.039,A -85,B 0,C 180,E1 11894.642,E2 11894.642} C_VEL
LIN {X 0,Y 473.235,Z 464.992,A -85,B 0,C 180,E1 11892.198,E2 11892.198} C_VEL
LIN {X 0,Y 470.532,Z 460.702,A -85,B 0,C 180,E1 11889.664,E2 11889.664} C_VEL
LIN {X 0,Y 467.611,Z 455.888,A -85,B 0,C 180,E1 11884.907,E2 11884.907} C_VEL
LIN {X 0,Y 467.323,Z 455.245,A -85,B 0,C 180,E1 11880.49,E2 11880.49} C_VEL
LIN {X 0,Y 469.357,Z 456.696,A -85,B 0,C 180,E1 11876.336,E2 11876.336} C_VEL
LIN {X 0,Y 473.995,Z 462.475,A -85,B 0,C 180,E1 11871.753,E2 11871.753} C_VEL
LIN {X 0,Y 478.237,Z 467.952,A -85,B 0,C 180,E1 11868.91,E2 11868.91} C_VEL
LIN {X 0,Y 482.63,Z 473.822,A -85,B 0,C 180,E1 11866.522,E2 11866.522} C_VEL
LIN {X 0,Y 486.414,Z 478.95,A -85,B 0,C 180,E1 11864.745,E2 11864.745} C_VEL
LIN {X 0,Y 492.221,Z 486.977,A -85,B 0,C 180,E1 11862.351,E2 11862.351} C_VEL
LIN {X 0,Y 500.056,Z 498.586,A -85,B 0,C 180,E1 11859.548,E2 11859.548} C_VEL
LIN {X 0,Y 507.828,Z 510.602,A -85,B 0,C 180,E1 11857.116,E2 11857.116} C_VEL
LIN {X 0,Y 510.738,Z 515.633,A -85,B 0,C 180,E1 11856.262,E2 11856.262} C_VEL
LIN {X 0,Y 495.623,Z 733.006,A -85,B 0,C 180,E1 11852.801,E2 11852.801} C_VEL
LIN {X 0,Y 489.062,Z 827.656,A -85,B 0,C 180,E1 11851.269,E2 11851.269} C_VEL
LIN {X 0,Y 485.812,Z 855.551,A -85,B 0,C 180,E1 11850.71,E2 11850.71} C_VEL
LIN {X 0,Y 481.732,Z 880.495,A -85,B 0,C 180,E1 11850.046,E2 11850.046} C_VEL
LIN {X 0,Y 477.665,Z 901.372,A -85,B 0,C 180,E1 11849.353,E2 11849.353} C_VEL
LIN {X 0,Y 472.926,Z 922.399,A -85,B 0,C 180,E1 11848.518,E2 11848.518} C_VEL
LIN {X 0,Y 466.389,Z 947.931,A -85,B 0,C 180,E1 11847.298,E2 11847.298} C_VEL
LIN {X 0,Y 459.376,Z 971.648,A -85,B 0,C 180,E1 11845.913,E2 11845.913} C_VEL
LIN {X 0,Y 453.166,Z 990.836,A -85,B 0,C 180,E1 11844.614,E2 11844.614} C_VEL
LIN {X 0,Y 446.399,Z 1010.315,A -85,B 0,C 180,E1 11843.095,E2 11843.095} C_VEL
LIN {X 0,Y 437.69,Z 1033.721,A -85,B 0,C 180,E1 11840.96,E2 11840.96} C_VEL
LIN {X 0,Y 429.999,Z 1053.018,A -85,B 0,C 180,E1 11838.885,E2 11838.885} C_VEL
LIN {X 0,Y 423.036,Z 1069.883,A -85,B 0,C 180,E1 11836.81,E2 11836.81} C_VEL
LIN {X 0,Y 415.433,Z 1087.943,A -85,B 0,C 180,E1 11834.265,E2 11834.265} C_VEL
LIN {X 0,Y 407.662,Z 1105.994,A -85,B 0,C 180,E1 11831.283,E2 11831.283} C_VEL
LIN {X 0,Y 401.506,Z 1120.289,A -85,B 0,C 180,E1 11828.558,E2 11828.558} C_VEL
LIN {X 0,Y 396.198,Z 1132.849,A -85,B 0,C 180,E1 11825.837,E2 11825.837} C_VEL
LIN {X 0,Y 390.777,Z 1146.318,A -85,B 0,C 180,E1 11822.501,E2 11822.501} C_VEL
LIN {X 0,Y 385.788,Z 1159.436,A -85,B 0,C 180,E1 11818.651,E2 11818.651} C_VEL
LIN {X 0,Y 382.677,Z 1168.533,A -85,B 0,C 180,E1 11815.538,E2 11815.538} C_VEL
LIN {X 0,Y 380.271,Z 1176.45,A -85,B 0,C 180,E1 11812.411,E2 11812.411} C_VEL
LIN {X 0,Y 378.492,Z 1183.242,A -85,B 0,C 180,E1 11809.282,E2 11809.282} C_VEL
LIN {X 0,Y 377.198,Z 1189.49,A -85,B 0,C 180,E1 11805.844,E2 11805.844} C_VEL
LIN {X 0,Y 376.331,Z 1195.285,A -85,B 0,C 180,E1 11801.805,E2 11801.805} C_VEL
LIN {X 0,Y 376.028,Z 1199.017,A -85,B 0,C 180,E1 11798.101,E2 11798.101} C_VEL
LIN {X 0,Y 375.952,Z 1201.169,A -85,B 0,C 180,E1 11794.882,E2 11794.882} C_VEL
LIN {X 0,Y 375.944,Z 1202.231,A -85,B 0,C 180,E1 11791.829,E2 11791.829} C_VEL
LIN {X 0,Y 375.945,Z 1202.35,A -85,B 0,C 180,E1 11788.933,E2 11788.933} C_VEL
LIN {X 0,Y 375.943,Z 1201.514,A -85,B 0,C 180,E1 11785.857,E2 11785.857} C_VEL
LIN {X 0,Y 375.993,Z 1199.732,A -85,B 0,C 180,E1 11782.82,E2 11782.82} C_VEL
LIN {X 0,Y 376.169,Z 1196.961,A -85,B 0,C 180,E1 11779.741,E2 11779.741} C_VEL
LIN {X 0,Y 376.585,Z 1193.198,A -85,B 0,C 180,E1 11776.644,E2 11776.644} C_VEL
LIN {X 0,Y 377.383,Z 1188.421,A -85,B 0,C 180,E1 11773.531,E2 11773.531} C_VEL
LIN {X 0,Y 378.649,Z 1182.6,A -85,B 0,C 180,E1 11770.405,E2 11770.405} C_VEL
LIN {X 0,Y 380.588,Z 1175.332,A -85,B 0,C 180,E1 11767.118,E2 11767.118} C_VEL
LIN {X 0,Y 383.84,Z 1165.134,A -85,B 0,C 180,E1 11763.214,E2 11763.214} C_VEL
LIN {X 0,Y 388.019,Z 1153.345,A -85,B 0,C 180,E1 11759.493,E2 11759.493} C_VEL
LIN {X 0,Y 392.145,Z 1142.74,A -85,B 0,C 180,E1 11756.581,E2 11756.581} C_VEL
LIN {X 0,Y 397.083,Z 1130.736,A -85,B 0,C 180,E1 11753.687,E2 11753.687} C_VEL
LIN {X 0,Y 403.835,Z 1114.913,A -85,B 0,C 180,E1 11750.357,E2 11750.357} C_VEL
LIN {X 0,Y 411.219,Z 1097.579,A -85,B 0,C 180,E1 11747.282,E2 11747.282} C_VEL
LIN {X 0,Y 417.808,Z 1082.179,A -85,B 0,C 180,E1 11744.897,E2 11744.897} C_VEL
LIN {X 0,Y 425.249,Z 1064.586,A -85,B 0,C 180,E1 11742.513,E2 11742.513} C_VEL
LIN {X 0,Y 434.074,Z 1042.813,A -85,B 0,C 180,E1 11739.992,E2 11739.992} C_VEL
LIN {X 0,Y 440.922,Z 1025.027,A -85,B 0,C 180,E1 11738.219,E2 11738.219} C_VEL
LIN {X 0,Y 447.642,Z 1006.637,A -85,B 0,C 180,E1 11736.612,E2 11736.612} C_VEL
LIN {X 0,Y 454.54,Z 986.547,A -85,B 0,C 180,E1 11735.084,E2 11735.084} C_VEL
LIN {X 0,Y 462.815,Z 959.992,A -85,B 0,C 180,E1 11733.383,E2 11733.383} C_VEL
LIN {X 0,Y 468.656,Z 938.985,A -85,B 0,C 180,E1 11732.259,E2 11732.259} C_VEL
LIN {X 0,Y 473.913,Z 917.883,A -85,B 0,C 180,E1 11731.297,E2 11731.297} C_VEL
LIN {X 0,Y 479.389,Z 892.842,A -85,B 0,C 180,E1 11730.348,E2 11730.348} C_VEL
LIN {X 0,Y 484.073,Z 866.106,A -85,B 0,C 180,E1 11729.558,E2 11729.558} C_VEL
LIN {X 0,Y 487.222,Z 843.769,A -85,B 0,C 180,E1 11729.045,E2 11729.045} C_VEL
LIN {X 0,Y 489.595,Z 820.372,A -85,B 0,C 180,E1 11728.612,E2 11728.612} C_VEL
LIN {X 0,Y 504.603,Z 601.274,A -85,B 0,C 180,E1 11725.106,E2 11725.106} C_VEL
LIN {X 0,Y 510.609,Z 515.29,A -85,B 0,C 180,E1 11723.729,E2 11723.729} C_VEL
LIN {X 0,Y 502.506,Z 502.378,A -85,B 0,C 180,E1 11721.293,E2 11721.293} C_VEL
LIN {X 0,Y 494.735,Z 490.745,A -85,B 0,C 180,E1 11718.653,E2 11718.653} C_VEL
LIN {X 0,Y 488.23,Z 481.446,A -85,B 0,C 180,E1 11716.111,E2 11716.111} C_VEL
LIN {X 0,Y 483.874,Z 475.583,A -85,B 0,C 180,E1 11714.174,E2 11714.174} C_VEL
LIN {X 0,Y 480.754,Z 471.415,A -85,B 0,C 180,E1 11712.614,E2 11712.614} C_VEL
LIN {X 0,Y 477.073,Z 466.516,A -85,B 0,C 180,E1 11710.506,E2 11710.506} C_VEL
LIN {X 0,Y 473.318,Z 461.687,A -85,B 0,C 180,E1 11707.892,E2 11707.892} C_VEL
LIN {X 0,Y 468.937,Z 456.299,A -85,B 0,C 180,E1 11703.423,E2 11703.423} C_VEL
LIN {X 0,Y 466.938,Z 454.991,A -85,B 0,C 180,E1 11698.896,E2 11698.896} C_VEL
LIN {X 0,Y 467.485,Z 455.841,A -85,B 0,C 180,E1 11694.6,E2 11694.6} C_VEL
LIN {X 0,Y 470.912,Z 461.425,A -85,B 0,C 180,E1 11689.602,E2 11689.602} C_VEL
LIN {X 0,Y 474.231,Z 466.621,A -85,B 0,C 180,E1 11686.775,E2 11686.775} C_VEL
LIN {X 0,Y 477.544,Z 471.536,A -85,B 0,C 180,E1 11684.579,E2 11684.579} C_VEL
LIN {X 0,Y 482.949,Z 479.661,A -85,B 0,C 180,E1 11681.657,E2 11681.657} C_VEL
LIN {X 0,Y 488.745,Z 488.742,A -85,B 0,C 180,E1 11679.053,E2 11679.053} C_VEL
LIN {X 0,Y 495.982,Z 500.404,A -85,B 0,C 180,E1 11676.285,E2 11676.285} C_VEL
LIN {X 0,Y 503.343,Z 512.848,A -85,B 0,C 180,E1 11673.832,E2 11673.832} C_VEL
LIN {X 0,Y 507.882,Z 520.938,A -85,B 0,C 180,E1 11672.451,E2 11672.451} C_VEL
LIN {X 0,Y 493,Z 747.269,A -85,B 0,C 180,E1 11668.989,E2 11668.989} C_VEL
LIN {X 0,Y 487.476,Z 831.63,A -85,B 0,C 180,E1 11667.679,E2 11667.679} C_VEL
LIN {X 0,Y 484.07,Z 860.519,A -85,B 0,C 180,E1 11667.098,E2 11667.098} C_VEL
LIN {X 0,Y 480.503,Z 882.243,A -85,B 0,C 180,E1 11666.524,E2 11666.524} C_VEL
LIN {X 0,Y 476.264,Z 903.801,A -85,B 0,C 180,E1 11665.81,E2 11665.81} C_VEL
LIN {X 0,Y 470.215,Z 929.714,A -85,B 0,C 180,E1 11664.741,E2 11664.741} C_VEL
LIN {X 0,Y 464.315,Z 951.223,A -85,B 0,C 180,E1 11663.648,E2 11663.648} C_VEL
LIN {X 0,Y 458.591,Z 970.036,A -85,B 0,C 180,E1 11662.527,E2 11662.527} C_VEL
LIN {X 0,Y 452.207,Z 989.174,A -85,B 0,C 180,E1 11661.207,E2 11661.207} C_VEL
LIN {X 0,Y 443.722,Z 1012.378,A -85,B 0,C 180,E1 11659.312,E2 11659.312} C_VEL
LIN {X 0,Y 436.666,Z 1030.141,A -85,B 0,C 180,E1 11657.601,E2 11657.601} C_VEL
LIN {X 0,Y 429.955,Z 1046.182,A -85,B 0,C 180,E1 11655.829,E2 11655.829} C_VEL
LIN {X 0,Y 422.162,Z 1064.101,A -85,B 0,C 180,E1 11653.551,E2 11653.551} C_VEL
LIN {X 0,Y 414.043,Z 1081.846,A -85,B 0,C 180,E1 11650.878,E2 11650.878} C_VEL
LIN {X 0,Y 407.755,Z 1095.334,A -85,B 0,C 180,E1 11648.525,E2 11648.525} C_VEL
LIN {X 0,Y 401.775,Z 1108.143,A -85,B 0,C 180,E1 11645.967,E2 11645.967} C_VEL
LIN {X 0,Y 395.052,Z 1122.771,A -85,B 0,C 180,E1 11642.559,E2 11642.559} C_VEL
LIN {X 0,Y 389.749,Z 1134.558,A -85,B 0,C 180,E1 11639.277,E2 11639.277} C_VEL
LIN {X 0,Y 385.696,Z 1144.191,A -85,B 0,C 180,E1 11636.149,E2 11636.149} C_VEL
LIN {X 0,Y 381.772,Z 1154.479,A -85,B 0,C 180,E1 11632.157,E2 11632.157} C_VEL
LIN {X 0,Y 379.305,Z 1161.89,A -85,B 0,C 180,E1 11628.601,E2 11628.601} C_VEL
LIN {X 0,Y 377.766,Z 1167.468,A -85,B 0,C 180,E1 11625.348,E2 11625.348} C_VEL
LIN {X 0,Y 376.679,Z 1172.726,A -85,B 0,C 180,E1 11621.484,E2 11621.484} C_VEL
LIN {X 0,Y 376.172,Z 1176.287,A -85,B 0,C 180,E1 11617.638,E2 11617.638} C_VEL
LIN {X 0,Y 376.005,Z 1178.196,A -85,B 0,C 180,E1 11614.423,E2 11614.423} C_VEL
LIN {X 0,Y 375.972,Z 1179.079,A -85,B 0,C 180,E1 11611.372,E2 11611.372} C_VEL
LIN {X 0,Y 375.976,Z 1179.05,A -85,B 0,C 180,E1 11608.324,E2 11608.324} C_VEL
LIN {X 0,Y 376.014,Z 1178.046,A -85,B 0,C 180,E1 11605.119,E2 11605.119} C_VEL
LIN {X 0,Y 376.271,Z 1175.585,A -85,B 0,C 180,E1 11601.288,E2 11601.288} C_VEL
LIN {X 0,Y 376.688,Z 1172.681,A -85,B 0,C 180,E1 11598.382,E2 11598.382} C_VEL
LIN {X 0,Y 375.947,Z 1171.339,A -85,B 0,C 180,E1 11597.224,E2 11597.224} C_VEL
LIN {X 0,Y 370.62,Z 1167.38,A -85,B 0,C 180,E1 11594.029,E2 11594.029} C_VEL
LIN {X 0,Y 370.398,Z 1166.014,A -85,B 0,C 180,E1 11593.105,E2 11593.105} C_VEL
LIN {X 0,Y 372.965,Z 1158.016,A -85,B 0,C 180,E1 11588.782,E2 11588.782} C_VEL
LIN {X 0,Y 375.822,Z 1150.457,A -85,B 0,C 180,E1 11585.479,E2 11585.479} C_VEL
LIN {X 0,Y 379.548,Z 1141.629,A -85,B 0,C 180,E1 11582.207,E2 11582.207} C_VEL
LIN {X 0,Y 385.163,Z 1129.296,A -85,B 0,C 180,E1 11578.373,E2 11578.373} C_VEL
LIN {X 0,Y 390.927,Z 1117.159,A -85,B 0,C 180,E1 11575.224,E2 11575.224} C_VEL
LIN {X 0,Y 396.961,Z 1104.75,A -85,B 0,C 180,E1 11572.443,E2 11572.443} C_VEL
LIN {X 0,Y 405.012,Z 1088.22,A -85,B 0,C 180,E1 11569.282,E2 11569.282} C_VEL
LIN {X 0,Y 412.62,Z 1072.209,A -85,B 0,C 180,E1 11566.704,E2 11566.704} C_VEL
LIN {X 0,Y 419.917,Z 1056.47,A -85,B 0,C 180,E1 11564.509,E2 11564.509} C_VEL
LIN {X 0,Y 429.011,Z 1035.969,A -85,B 0,C 180,E1 11562.072,E2 11562.072} C_VEL
LIN {X 0,Y 436.59,Z 1017.63,A -85,B 0,C 180,E1 11560.229,E2 11560.229} C_VEL
LIN {X 0,Y 443.356,Z 1000.219,A -85,B 0,C 180,E1 11558.711,E2 11558.711} C_VEL
LIN {X 0,Y 451.37,Z 978.07,A -85,B 0,C 180,E1 11557.053,E2 11557.053} C_VEL
LIN {X 0,Y 458.776,Z 954.825,A -85,B 0,C 180,E1 11555.617,E2 11555.617} C_VEL
LIN {X 0,Y 464.487,Z 934.876,A -85,B 0,C 180,E1 11554.575,E2 11554.575} C_VEL
LIN {X 0,Y 470.057,Z 913,A -85,B 0,C 180,E1 11553.616,E2 11553.616} C_VEL
LIN {X 0,Y 475.728,Z 886.184,A -85,B 0,C 180,E1 11552.674,E2 11552.674} C_VEL
LIN {X 0,Y 479.368,Z 865.153,A -85,B 0,C 180,E1 11552.095,E2 11552.095} C_VEL
LIN {X 0,Y 482.322,Z 843.553,A -85,B 0,C 180,E1 11551.621,E2 11551.621} C_VEL
LIN {X 0,Y 484.904,Z 814.903,A -85,B 0,C 180,E1 11551.128,E2 11551.128} C_VEL
LIN {X 0,Y 500.035,Z 586.472,A -85,B 0,C 180,E1 11547.628,E2 11547.628} C_VEL
LIN {X 0,Y 504.269,Z 525.45,A -85,B 0,C 180,E1 11546.687,E2 11546.687} C_VEL
LIN {X 0,Y 497.402,Z 513.425,A -85,B 0,C 180,E1 11544.463,E2 11544.463} C_VEL
LIN {X 0,Y 491.143,Z 502.896,A -85,B 0,C 180,E1 11542.188,E2 11542.188} C_VEL
LIN {X 0,Y 485.461,Z 493.654,A -85,B 0,C 180,E1 11539.836,E2 11539.836} C_VEL
LIN {X 0,Y 480.021,Z 485.066,A -85,B 0,C 180,E1 11537.205,E2 11537.205} C_VEL
LIN {X 0,Y 475.128,Z 477.513,A -85,B 0,C 180,E1 11534.316,E2 11534.316} C_VEL
LIN {X 0,Y 471.967,Z 472.702,A -85,B 0,C 180,E1 11531.983,E2 11531.983} C_VEL
LIN {X 0,Y 469.338,Z 468.473,A -85,B 0,C 180,E1 11529.442,E2 11529.442} C_VEL
LIN {X 0,Y 466.596,Z 463.792,A -85,B 0,C 180,E1 11524.794,E2 11524.794} C_VEL
LIN {X 0,Y 466.348,Z 463.186,A -85,B 0,C 180,E1 11520.491,E2 11520.491} C_VEL
LIN {X 0,Y 468.288,Z 464.57,A -85,B 0,C 180,E1 11516.45,E2 11516.45} C_VEL
LIN {X 0,Y 472.843,Z 470.408,A -85,B 0,C 180,E1 11511.855,E2 11511.855} C_VEL
LIN {X 0,Y 476.849,Z 475.64,A -85,B 0,C 180,E1 11509.122,E2 11509.122} C_VEL
LIN {X 0,Y 481.053,Z 481.352,A -85,B 0,C 180,E1 11506.783,E2 11506.783} C_VEL
LIN {X 0,Y 484.889,Z 486.669,A -85,B 0,C 180,E1 11504.94,E2 11504.94} C_VEL
LIN {X 0,Y 490.406,Z 494.445,A -85,B 0,C 180,E1 11502.62,E2 11502.62} C_VEL
LIN {X 0,Y 498.126,Z 506.067,A -85,B 0,C 180,E1 11499.802,E2 11499.802} C_VEL
LIN {X 0,Y 505.616,Z 517.923,A -85,B 0,C 180,E1 11497.409,E2 11497.409} C_VEL
LIN {X 0,Y 506.934,Z 520.444,A -85,B 0,C 180,E1 11497.002,E2 11497.002} C_VEL
LIN {X 0,Y 491.395,Z 738.333,A -85,B 0,C 180,E1 11493.533,E2 11493.533} C_VEL
LIN {X 0,Y 485.005,Z 827.857,A -85,B 0,C 180,E1 11492.081,E2 11492.081} C_VEL
LIN {X 0,Y 481.644,Z 855.938,A -85,B 0,C 180,E1 11491.519,E2 11491.519} C_VEL
LIN {X 0,Y 477.502,Z 880.677,A -85,B 0,C 180,E1 11490.861,E2 11490.861} C_VEL
LIN {X 0,Y 473.386,Z 901.34,A -85,B 0,C 180,E1 11490.178,E2 11490.178} C_VEL
LIN {X 0,Y 468.773,Z 921.371,A -85,B 0,C 180,E1 11489.389,E2 11489.389} C_VEL
LIN {X 0,Y 462.891,Z 944.023,A -85,B 0,C 180,E1 11488.327,E2 11488.327} C_VEL
LIN {X 0,Y 455.323,Z 969.49,A -85,B 0,C 180,E1 11486.882,E2 11486.882} C_VEL
LIN {X 0,Y 448.573,Z 989.876,A -85,B 0,C 180,E1 11485.516,E2 11485.516} C_VEL
LIN {X 0,Y 441.716,Z 1009.133,A -85,B 0,C 180,E1 11484.022,E2 11484.022} C_VEL
LIN {X 0,Y 433.249,Z 1031.449,A -85,B 0,C 180,E1 11482.014,E2 11482.014} C_VEL
LIN {X 0,Y 424.517,Z 1052.649,A -85,B 0,C 180,E1 11479.74,E2 11479.74} C_VEL
LIN {X 0,Y 417.459,Z 1069.195,A -85,B 0,C 180,E1 11477.697,E2 11477.697} C_VEL
LIN {X 0,Y 410.229,Z 1085.7,A -85,B 0,C 180,E1 11475.374,E2 11475.374} C_VEL
LIN {X 0,Y 401.335,Z 1105.673,A -85,B 0,C 180,E1 11472.081,E2 11472.081} C_VEL
LIN {X 0,Y 395.146,Z 1119.468,A -85,B 0,C 180,E1 11469.429,E2 11469.429} C_VEL
LIN {X 0,Y 389.668,Z 1131.888,A -85,B 0,C 180,E1 11466.717,E2 11466.717} C_VEL
LIN {X 0,Y 384.38,Z 1144.239,A -85,B 0,C 180,E1 11463.646,E2 11463.646} C_VEL
LIN {X 0,Y 378.805,Z 1158.197,A -85,B 0,C 180,E1 11459.577,E2 11459.577} C_VEL
LIN {X 0,Y 375.106,Z 1168.326,A -85,B 0,C 180,E1 11456.062,E2 11456.062} C_VEL
LIN {X 0,Y 372.578,Z 1176.173,A -85,B 0,C 180,E1 11452.9,E2 11452.9} C_VEL
LIN {X 0,Y 370.691,Z 1182.971,A -85,B 0,C 180,E1 11449.704,E2 11449.704} C_VEL
LIN {X 0,Y 369.296,Z 1189.225,A -85,B 0,C 180,E1 11446.193,E2 11446.193} C_VEL
LIN {X 0,Y 368.367,Z 1195.029,A -85,B 0,C 180,E1 11442.064,E2 11442.064} C_VEL
LIN {X 0,Y 368.036,Z 1198.765,A -85,B 0,C 180,E1 11438.278,E2 11438.278} C_VEL
LIN {X 0,Y 367.955,Z 1200.92,A -85,B 0,C 180,E1 11434.988,E2 11434.988} C_VEL
LIN {X 0,Y 367.947,Z 1201.96,A -85,B 0,C 180,E1 11432.024,E2 11432.024} C_VEL
LIN {X 0,Y 367.949,Z 1202.103,A -85,B 0,C 180,E1 11428.91,E2 11428.91} C_VEL
LIN {X 0,Y 367.946,Z 1201.277,A -85,B 0,C 180,E1 11425.792,E2 11425.792} C_VEL
LIN {X 0,Y 368.006,Z 1199.451,A -85,B 0,C 180,E1 11422.626,E2 11422.626} C_VEL
LIN {X 0,Y 368.195,Z 1196.626,A -85,B 0,C 180,E1 11419.442,E2 11419.442} C_VEL
LIN {X 0,Y 368.643,Z 1192.937,A -85,B 0,C 180,E1 11416.351,E2 11416.351} C_VEL
LIN {X 0,Y 369.488,Z 1188.153,A -85,B 0,C 180,E1 11413.168,E2 11413.168} C_VEL
LIN {X 0,Y 370.856,Z 1182.327,A -85,B 0,C 180,E1 11409.976,E2 11409.976} C_VEL
LIN {X 0,Y 372.908,Z 1175.053,A -85,B 0,C 180,E1 11406.619,E2 11406.619} C_VEL
LIN {X 0,Y 376.363,Z 1164.844,A -85,B 0,C 180,E1 11402.638,E2 11402.638} C_VEL
LIN {X 0,Y 380.772,Z 1153.048,A -85,B 0,C 180,E1 11398.848,E2 11398.848} C_VEL
LIN {X 0,Y 385.125,Z 1142.437,A -85,B 0,C 180,E1 11395.889,E2 11395.889} C_VEL
LIN {X 0,Y 390.241,Z 1130.543,A -85,B 0,C 180,E1 11392.978,E2 11392.978} C_VEL
LIN {X 0,Y 397.116,Z 1115.091,A -85,B 0,C 180,E1 11389.677,E2 11389.677} C_VEL
LIN {X 0,Y 404.771,Z 1097.867,A -85,B 0,C 180,E1 11386.574,E2 11386.574} C_VEL
LIN {X 0,Y 411.475,Z 1082.781,A -85,B 0,C 180,E1 11384.205,E2 11384.205} C_VEL
LIN {X 0,Y 418.501,Z 1066.719,A -85,B 0,C 180,E1 11381.989,E2 11381.989} C_VEL
LIN {X 0,Y 427.453,Z 1045.646,A -85,B 0,C 180,E1 11379.473,E2 11379.473} C_VEL
LIN {X 0,Y 435.569,Z 1025.225,A -85,B 0,C 180,E1 11377.414,E2 11377.414} C_VEL
LIN {X 0,Y 442.53,Z 1006.734,A -85,B 0,C 180,E1 11375.792,E2 11375.792} C_VEL
LIN {X 0,Y 449.822,Z 986.072,A -85,B 0,C 180,E1 11374.219,E2 11374.219} C_VEL
LIN {X 0,Y 458.023,Z 960.452,A -85,B 0,C 180,E1 11372.579,E2 11372.579} C_VEL
LIN {X 0,Y 464.089,Z 939.198,A -85,B 0,C 180,E1 11371.44,E2 11371.44} C_VEL
LIN {X 0,Y 469.386,Z 918.485,A -85,B 0,C 180,E1 11370.496,E2 11370.496} C_VEL
LIN {X 0,Y 474.494,Z 895.775,A -85,B 0,C 180,E1 11369.629,E2 11369.629} C_VEL
LIN {X 0,Y 479.715,Z 867.463,A -85,B 0,C 180,E1 11368.774,E2 11368.774} C_VEL
LIN {X 0,Y 483.03,Z 844.649,A -85,B 0,C 180,E1 11368.246,E2 11368.246} C_VEL
LIN {X 0,Y 485.426,Z 821.94,A -85,B 0,C 180,E1 11367.823,E2 11367.823} C_VEL
LIN {X 0,Y 500.651,Z 605.923,A -85,B 0,C 180,E1 11364.362,E2 11364.362} C_VEL
LIN {X 0,Y 506.821,Z 520.116,A -85,B 0,C 180,E1 11362.994,E2 11362.994} C_VEL
LIN {X 0,Y 498.978,Z 507.392,A -85,B 0,C 180,E1 11360.529,E2 11360.529} C_VEL
LIN {X 0,Y 490.892,Z 495.33,A -85,B 0,C 180,E1 11357.637,E2 11357.637} C_VEL
LIN {X 0,Y 485.36,Z 487.42,A -85,B 0,C 180,E1 11355.351,E2 11355.351} C_VEL
LIN {X 0,Y 482.148,Z 482.96,A -85,B 0,C 180,E1 11353.859,E2 11353.859} C_VEL
LIN {X 0,Y 479.207,Z 478.97,A -85,B 0,C 180,E1 11352.349,E2 11352.349} C_VEL
LIN {X 0,Y 475.701,Z 474.209,A -85,B 0,C 180,E1 11350.292,E2 11350.292} C_VEL
LIN {X 0,Y 472.025,Z 469.433,A -85,B 0,C 180,E1 11347.669,E2 11347.669} C_VEL
LIN {X 0,Y 467.959,Z 464.251,A -85,B 0,C 180,E1 11343.43,E2 11343.43} C_VEL
LIN {X 0,Y 465.982,Z 462.936,A -85,B 0,C 180,E1 11339.016,E2 11339.016} C_VEL
LIN {X 0,Y 466.468,Z 463.741,A -85,B 0,C 180,E1 11334.711,E2 11334.711} C_VEL
LIN {X 0,Y 469.759,Z 469.24,A -85,B 0,C 180,E1 11329.762,E2 11329.762} C_VEL
LIN {X 0,Y 472.933,Z 474.322,A -85,B 0,C 180,E1 11326.987,E2 11326.987} C_VEL
LIN {X 0,Y 476.182,Z 479.258,A -85,B 0,C 180,E1 11324.783,E2 11324.783} C_VEL
LIN {X 0,Y 481.324,Z 487.14,A -85,B 0,C 180,E1 11321.938,E2 11321.938} C_VEL
LIN {X 0,Y 486.952,Z 496.129,A -85,B 0,C 180,E1 11319.349,E2 11319.349} C_VEL
LIN {X 0,Y 493.914,Z 507.573,A -85,B 0,C 180,E1 11316.622,E2 11316.622} C_VEL
LIN {X 0,Y 501.066,Z 519.896,A -85,B 0,C 180,E1 11314.181,E2 11314.181} C_VEL
LIN {X 0,Y 504.147,Z 525.695,A -85,B 0,C 180,E1 11313.204,E2 11313.204} C_VEL
LIN {X 0,Y 488.934,Z 750.616,A -85,B 0,C 180,E1 11309.76,E2 11309.76} C_VEL
LIN {X 0,Y 483.462,Z 831.645,A -85,B 0,C 180,E1 11308.499,E2 11308.499} C_VEL
LIN {X 0,Y 479.972,Z 860.559,A -85,B 0,C 180,E1 11307.918,E2 11307.918} C_VEL
LIN {X 0,Y 476.306,Z 882.365,A -85,B 0,C 180,E1 11307.346,E2 11307.346} C_VEL
LIN {X 0,Y 471.99,Z 903.833,A -85,B 0,C 180,E1 11306.636,E2 11306.636} C_VEL
LIN {X 0,Y 465.954,Z 929.184,A -85,B 0,C 180,E1 11305.598,E2 11305.598} C_VEL
LIN {X 0,Y 459.604,Z 951.756,A -85,B 0,C 180,E1 11304.454,E2 11304.454} C_VEL
LIN {X 0,Y 453.702,Z 970.633,A -85,B 0,C 180,E1 11303.327,E2 11303.327} C_VEL
LIN {X 0,Y 446.911,Z 990.422,A -85,B 0,C 180,E1 11301.956,E2 11301.956} C_VEL
LIN {X 0,Y 438.204,Z 1013.423,A -85,B 0,C 180,E1 11300.056,E2 11300.056} C_VEL
LIN {X 0,Y 431.211,Z 1030.509,A -85,B 0,C 180,E1 11298.401,E2 11298.401} C_VEL
LIN {X 0,Y 424.093,Z 1047.002,A -85,B 0,C 180,E1 11296.566,E2 11296.566} C_VEL
LIN {X 0,Y 415.861,Z 1065.329,A -85,B 0,C 180,E1 11294.208,E2 11294.208} C_VEL
LIN {X 0,Y 407.702,Z 1082.474,A -85,B 0,C 180,E1 11291.581,E2 11291.581} C_VEL
LIN {X 0,Y 400.973,Z 1096.391,A -85,B 0,C 180,E1 11289.116,E2 11289.116} C_VEL
LIN {X 0,Y 393.841,Z 1111.169,A -85,B 0,C 180,E1 11286.086,E2 11286.086} C_VEL
LIN {X 0,Y 387.038,Z 1125.24,A -85,B 0,C 180,E1 11282.626,E2 11282.626} C_VEL
LIN {X 0,Y 382.194,Z 1135.645,A -85,B 0,C 180,E1 11279.634,E2 11279.634} C_VEL
LIN {X 0,Y 377.42,Z 1146.681,A -85,B 0,C 180,E1 11275.921,E2 11275.921} C_VEL
LIN {X 0,Y 373.636,Z 1156.103,A -85,B 0,C 180,E1 11272.003,E2 11272.003} C_VEL
LIN {X 0,Y 371.363,Z 1162.734,A -85,B 0,C 180,E1 11268.688,E2 11268.688} C_VEL
LIN {X 0,Y 369.62,Z 1168.945,A -85,B 0,C 180,E1 11264.892,E2 11264.892} C_VEL
LIN {X 0,Y 368.551,Z 1173.911,A -85,B 0,C 180,E1 11260.79,E2 11260.79} C_VEL
LIN {X 0,Y 368.165,Z 1176.752,A -85,B 0,C 180,E1 11257.491,E2 11257.491} C_VEL
LIN {X 0,Y 368.009,Z 1178.526,A -85,B 0,C 180,E1 11254.323,E2 11254.323} C_VEL
LIN {X 0,Y 367.977,Z 1179.347,A -85,B 0,C 180,E1 11251.246,E2 11251.246} C_VEL
LIN {X 0,Y 367.981,Z 1179.276,A -85,B 0,C 180,E1 11248.132,E2 11248.132} C_VEL
LIN {X 0,Y 368.038,Z 1178.165,A -85,B 0,C 180,E1 11244.7,E2 11244.7} C_VEL
LIN {X 0,Y 368.344,Z 1175.379,A -85,B 0,C 180,E1 11240.627,E2 11240.627} C_VEL
LIN {X 0,Y 369.013,Z 1171.527,A -85,B 0,C 180,E1 11237.004,E2 11237.004} C_VEL
LIN {X 0,Y 370.131,Z 1166.906,A -85,B 0,C 180,E1 11233.684,E2 11233.684} C_VEL
LIN {X 0,Y 370.398,Z 1166.014,A -85,B 0,C 180,E1 11233.105,E2 11233.105} C_VEL
LIN {X 0,Y 369.997,Z 1164.241,A -85,B 0,C 180,E1 11231.937,E2 11231.937} C_VEL
LIN {X 0,Y 365.654,Z 1159.019,A -85,B 0,C 180,E1 11228.706,E2 11228.706} C_VEL
LIN {X 0,Y 365.722,Z 1157.168,A -85,B 0,C 180,E1 11227.79,E2 11227.79} C_VEL
LIN {X 0,Y 368.838,Z 1149.551,A -85,B 0,C 180,E1 11224.467,E2 11224.467} C_VEL
LIN {X 0,Y 373.772,Z 1138.708,A -85,B 0,C 180,E1 11220.514,E2 11220.514} C_VEL
LIN {X 0,Y 379.226,Z 1127.348,A -85,B 0,C 180,E1 11217.102,E2 11217.102} C_VEL
LIN {X 0,Y 384.971,Z 1115.841,A -85,B 0,C 180,E1 11214.132,E2 11214.132} C_VEL
LIN {X 0,Y 392.599,Z 1100.888,A -85,B 0,C 180,E1 11210.831,E2 11210.831} C_VEL
LIN {X 0,Y 400.324,Z 1085.422,A -85,B 0,C 180,E1 11207.982,E2 11207.982} C_VEL
LIN {X 0,Y 407.127,Z 1071.618,A -85,B 0,C 180,E1 11205.775,E2 11205.775} C_VEL
LIN {X 0,Y 414.94,Z 1055.305,A -85,B 0,C 180,E1 11203.505,E2 11203.505} C_VEL
LIN {X 0,Y 424.355,Z 1034.535,A -85,B 0,C 180,E1 11201.063,E2 11201.063} C_VEL
LIN {X 0,Y 431.732,Z 1017.174,A -85,B 0,C 180,E1 11199.328,E2 11199.328} C_VEL
LIN {X 0,Y 438.658,Z 999.806,A -85,B 0,C 180,E1 11197.819,E2 11197.819} C_VEL
LIN {X 0,Y 446.691,Z 978.145,A -85,B 0,C 180,E1 11196.202,E2 11196.202} C_VEL
LIN {X 0,Y 454.145,Z 955.34,A -85,B 0,C 180,E1 11194.793,E2 11194.793} C_VEL
LIN {X 0,Y 459.988,Z 935.45,A -85,B 0,C 180,E1 11193.753,E2 11193.753} C_VEL
LIN {X 0,Y 465.364,Z 914.922,A -85,B 0,C 180,E1 11192.85,E2 11192.85} C_VEL
LIN {X 0,Y 471.167,Z 888.787,A -85,B 0,C 180,E1 11191.914,E2 11191.914} C_VEL
LIN {X 0,Y 475.199,Z 866.217,A -85,B 0,C 180,E1 11191.285,E2 11191.285} C_VEL
LIN {X 0,Y 478.216,Z 844.902,A -85,B 0,C 180,E1 11190.813,E2 11190.813} C_VEL
LIN {X 0,Y 480.774,Z 818.813,A -85,B 0,C 180,E1 11190.354,E2 11190.354} C_VEL
LIN {X 0,Y 496.467,Z 588.691,A -85,B 0,C 180,E1 11186.826,E2 11186.826} C_VEL
LIN {X 0,Y 500.592,Z 530.018,A -85,B 0,C 180,E1 11185.909,E2 11185.909} C_VEL
LIN {X 0,Y 493.817,Z 517.955,A -85,B 0,C 180,E1 11183.604,E2 11183.604} C_VEL
LIN {X 0,Y 487.14,Z 506.56,A -85,B 0,C 180,E1 11181.02,E2 11181.02} C_VEL
LIN {X 0,Y 481.56,Z 497.589,A -85,B 0,C 180,E1 11178.523,E2 11178.523} C_VEL
LIN {X 0,Y 477.239,Z 490.537,A -85,B 0,C 180,E1 11176.243,E2 11176.243} C_VEL
LIN {X 0,Y 473.617,Z 484.981,A -85,B 0,C 180,E1 11173.989,E2 11173.989} C_VEL
LIN {X 0,Y 470.705,Z 480.412,A -85,B 0,C 180,E1 11171.767,E2 11171.767} C_VEL
LIN {X 0,Y 468.261,Z 476.356,A -85,B 0,C 180,E1 11169.34,E2 11169.34} C_VEL
LIN {X 0,Y 465.583,Z 471.698,A -85,B 0,C 180,E1 11164.681,E2 11164.681} C_VEL
LIN {X 0,Y 465.401,Z 471.143,A -85,B 0,C 180,E1 11160.369,E2 11160.369} C_VEL
LIN {X 0,Y 467.301,Z 472.591,A -85,B 0,C 180,E1 11156.442,E2 11156.442} C_VEL
LIN {X 0,Y 471.625,Z 478.213,A -85,B 0,C 180,E1 11152.018,E2 11152.018} C_VEL
LIN {X 0,Y 475.558,Z 483.481,A -85,B 0,C 180,E1 11149.276,E2 11149.276} C_VEL
LIN {X 0,Y 479.592,Z 489.05,A -85,B 0,C 180,E1 11146.987,E2 11146.987} C_VEL
LIN {X 0,Y 483.493,Z 494.567,A -85,B 0,C 180,E1 11145.08,E2 11145.08} C_VEL
LIN {X 0,Y 488.88,Z 502.364,A -85,B 0,C 180,E1 11142.779,E2 11142.779} C_VEL
LIN {X 0,Y 496.61,Z 514.136,A -85,B 0,C 180,E1 11139.922,E2 11139.922} C_VEL
LIN {X 0,Y 503.249,Z 524.935,A -85,B 0,C 180,E1 11137.759,E2 11137.759} C_VEL
LIN {X 0,Y 487.279,Z 743.222,A -85,B 0,C 180,E1 11134.285,E2 11134.285} C_VEL
LIN {X 0,Y 481.038,Z 828.165,A -85,B 0,C 180,E1 11132.906,E2 11132.906} C_VEL
LIN {X 0,Y 477.536,Z 856.552,A -85,B 0,C 180,E1 11132.336,E2 11132.336} C_VEL
LIN {X 0,Y 473.392,Z 880.758,A -85,B 0,C 180,E1 11131.695,E2 11131.695} C_VEL
LIN {X 0,Y 469.207,Z 901.315,A -85,B 0,C 180,E1 11131.017,E2 11131.017} C_VEL
LIN {X 0,Y 464.193,Z 922.539,A -85,B 0,C 180,E1 11130.182,E2 11130.182} C_VEL
LIN {X 0,Y 457.376,Z 947.892,A -85,B 0,C 180,E1 11128.976,E2 11128.976} C_VEL
LIN {X 0,Y 450.21,Z 970.944,A -85,B 0,C 180,E1 11127.639,E2 11127.639} C_VEL
LIN {X 0,Y 443.46,Z 990.736,A -85,B 0,C 180,E1 11126.303,E2 11126.303} C_VEL
LIN {X 0,Y 436.259,Z 1010.351,A -85,B 0,C 180,E1 11124.769,E2 11124.769} C_VEL
LIN {X 0,Y 426.808,Z 1034.197,A -85,B 0,C 180,E1 11122.576,E2 11122.576} C_VEL
LIN {X 0,Y 418.89,Z 1052.853,A -85,B 0,C 180,E1 11120.55,E2 11120.55} C_VEL
LIN {X 0,Y 411.706,Z 1069.147,A -85,B 0,C 180,E1 11118.523,E2 11118.523} C_VEL
LIN {X 0,Y 404.111,Z 1085.882,A -85,B 0,C 180,E1 11116.147,E2 11116.147} C_VEL
LIN {X 0,Y 395.085,Z 1105.355,A -85,B 0,C 180,E1 11112.904,E2 11112.904} C_VEL
LIN {X 0,Y 388.3,Z 1119.879,A -85,B 0,C 180,E1 11110.072,E2 11110.072} C_VEL
LIN {X 0,Y 382.325,Z 1132.895,A -85,B 0,C 180,E1 11107.165,E2 11107.165} C_VEL
LIN {X 0,Y 375.895,Z 1147.445,A -85,B 0,C 180,E1 11103.409,E2 11103.409} C_VEL
LIN {X 0,Y 370.91,Z 1159.34,A -85,B 0,C 180,E1 11099.736,E2 11099.736} C_VEL
LIN {X 0,Y 367.411,Z 1168.542,A -85,B 0,C 180,E1 11096.445,E2 11096.445} C_VEL
LIN {X 0,Y 364.787,Z 1176.266,A -85,B 0,C 180,E1 11093.247,E2 11093.247} C_VEL
LIN {X 0,Y 362.648,Z 1183.65,A -85,B 0,C 180,E1 11089.656,E2 11089.656} C_VEL
LIN {X 0,Y 361.02,Z 1190.948,A -85,B 0,C 180,E1 11085.254,E2 11085.254} C_VEL
LIN {X 0,Y 360.288,Z 1195.614,A -85,B 0,C 180,E1 11081.526,E2 11081.526} C_VEL
LIN {X 0,Y 360.038,Z 1198.633,A -85,B 0,C 180,E1 11078.303,E2 11078.303} C_VEL
LIN {X 0,Y 359.959,Z 1200.671,A -85,B 0,C 180,E1 11075.099,E2 11075.099} C_VEL
LIN {X 0,Y 359.951,Z 1201.713,A -85,B 0,C 180,E1 11072.069,E2 11072.069} C_VEL
LIN {X 0,Y 359.953,Z 1201.856,A -85,B 0,C 180,E1 11068.885,E2 11068.885} C_VEL
LIN {X 0,Y 359.949,Z 1201.028,A -85,B 0,C 180,E1 11065.698,E2 11065.698} C_VEL
LIN {X 0,Y 360.011,Z 1199.228,A -85,B 0,C 180,E1 11062.499,E2 11062.499} C_VEL
LIN {X 0,Y 360.208,Z 1196.448,A -85,B 0,C 180,E1 11059.281,E2 11059.281} C_VEL
LIN {X 0,Y 360.725,Z 1192.576,A -85,B 0,C 180,E1 11055.97,E2 11055.97} C_VEL
LIN {X 0,Y 361.608,Z 1187.887,A -85,B 0,C 180,E1 11052.79,E2 11052.79} C_VEL
LIN {X 0,Y 363.131,Z 1181.854,A -85,B 0,C 180,E1 11049.424,E2 11049.424} C_VEL
LIN {X 0,Y 365.517,Z 1174.04,A -85,B 0,C 180,E1 11045.774,E2 11045.774} C_VEL
LIN {X 0,Y 369.615,Z 1162.653,A -85,B 0,C 180,E1 11041.391,E2 11041.391} C_VEL
LIN {X 0,Y 373.872,Z 1152.063,A -85,B 0,C 180,E1 11037.973,E2 11037.973} C_VEL
LIN {X 0,Y 378.683,Z 1140.951,A -85,B 0,C 180,E1 11034.857,E2 11034.857} C_VEL
LIN {X 0,Y 385.363,Z 1126.303,A -85,B 0,C 180,E1 11031.295,E2 11031.295} C_VEL
LIN {X 0,Y 392.86,Z 1110.051,A -85,B 0,C 180,E1 11027.981,E2 11027.981} C_VEL
LIN {X 0,Y 399.372,Z 1096.042,A -85,B 0,C 180,E1 11025.491,E2 11025.491} C_VEL
LIN {X 0,Y 406.159,Z 1081.326,A -85,B 0,C 180,E1 11023.188,E2 11023.188} C_VEL
LIN {X 0,Y 414.307,Z 1063.354,A -85,B 0,C 180,E1 11020.729,E2 11020.729} C_VEL
LIN {X 0,Y 423.44,Z 1042.148,A -85,B 0,C 180,E1 11018.266,E2 11018.266} C_VEL
LIN {X 0,Y 430.547,Z 1024.812,A -85,B 0,C 180,E1 11016.531,E2 11016.531} C_VEL
LIN {X 0,Y 437.507,Z 1006.851,A -85,B 0,C 180,E1 11014.954,E2 11014.954} C_VEL
LIN {X 0,Y 444.619,Z 987.255,A -85,B 0,C 180,E1 11013.455,E2 11013.455} C_VEL
LIN {X 0,Y 453.021,Z 961.933,A -85,B 0,C 180,E1 11011.815,E2 11011.815} C_VEL
LIN {X 0,Y 459.658,Z 939.266,A -85,B 0,C 180,E1 11010.599,E2 11010.599} C_VEL
LIN {X 0,Y 464.953,Z 919.091,A -85,B 0,C 180,E1 11009.68,E2 11009.68} C_VEL
LIN {X 0,Y 470.007,Z 897.227,A -85,B 0,C 180,E1 11008.843,E2 11008.843} C_VEL
LIN {X 0,Y 475.448,Z 868.852,A -85,B 0,C 180,E1 11007.976,E2 11007.976} C_VEL
LIN {X 0,Y 478.976,Z 845.212,A -85,B 0,C 180,E1 11007.427,E2 11007.427} C_VEL
LIN {X 0,Y 481.426,Z 822.678,A -85,B 0,C 180,E1 11007.006,E2 11007.006} C_VEL
LIN {X 0,Y 496.918,Z 608.733,A -85,B 0,C 180,E1 11003.578,E2 11003.578} C_VEL
LIN {X 0,Y 503.039,Z 524.712,A -85,B 0,C 180,E1 11002.22,E2 11002.22} C_VEL
LIN {X 0,Y 495.674,Z 512.852,A -85,B 0,C 180,E1 10999.81,E2 10999.81} C_VEL
LIN {X 0,Y 488.108,Z 501.203,A -85,B 0,C 180,E1 10996.973,E2 10996.973} C_VEL
LIN {X 0,Y 481.51,Z 491.694,A -85,B 0,C 180,E1 10994.061,E2 10994.061} C_VEL
LIN {X 0,Y 477.667,Z 486.522,A -85,B 0,C 180,E1 10992.083,E2 10992.083} C_VEL
LIN {X 0,Y 474.335,Z 481.902,A -85,B 0,C 180,E1 10990.077,E2 10990.077} C_VEL
LIN {X 0,Y 470.741,Z 477.174,A -85,B 0,C 180,E1 10987.445,E2 10987.445} C_VEL
LIN {X 0,Y 466.891,Z 472.145,A -85,B 0,C 180,E1 10983.315,E2 10983.315} C_VEL
LIN {X 0,Y 464.988,Z 470.872,A -85,B 0,C 180,E1 10978.891,E2 10978.891} C_VEL
LIN {X 0,Y 465.499,Z 471.7,A -85,B 0,C 180,E1 10974.7,E2 10974.7} C_VEL
LIN {X 0,Y 468.665,Z 477.168,A -85,B 0,C 180,E1 10969.862,E2 10969.862} C_VEL
LIN {X 0,Y 471.718,Z 482.164,A -85,B 0,C 180,E1 10967.14,E2 10967.14} C_VEL
LIN {X 0,Y 474.822,Z 486.979,A -85,B 0,C 180,E1 10964.988,E2 10964.988} C_VEL
LIN {X 0,Y 479.714,Z 494.62,A -85,B 0,C 180,E1 10962.22,E2 10962.22} C_VEL
LIN {X 0,Y 485.172,Z 503.515,A -85,B 0,C 180,E1 10959.649,E2 10959.649} C_VEL
LIN {X 0,Y 491.863,Z 514.741,A -85,B 0,C 180,E1 10956.963,E2 10956.963} C_VEL
LIN {X 0,Y 498.726,Z 526.793,A -85,B 0,C 180,E1 10954.561,E2 10954.561} C_VEL
LIN {X 0,Y 500.513,Z 530.369,A -85,B 0,C 180,E1 10953.968,E2 10953.968} C_VEL
LIN {X 0,Y 484.99,Z 753.563,A -85,B 0,C 180,E1 10950.551,E2 10950.551} C_VEL
LIN {X 0,Y 479.539,Z 831.768,A -85,B 0,C 180,E1 10949.331,E2 10949.331} C_VEL
LIN {X 0,Y 475.969,Z 860.621,A -85,B 0,C 180,E1 10948.753,E2 10948.753} C_VEL
LIN {X 0,Y 472.211,Z 882.483,A -85,B 0,C 180,E1 10948.182,E2 10948.182} C_VEL
LIN {X 0,Y 467.817,Z 903.863,A -85,B 0,C 180,E1 10947.477,E2 10947.477} C_VEL
LIN {X 0,Y 461.803,Z 928.654,A -85,B 0,C 180,E1 10946.469,E2 10946.469} C_VEL
LIN {X 0,Y 455.317,Z 951.214,A -85,B 0,C 180,E1 10945.335,E2 10945.335} C_VEL
LIN {X 0,Y 449.567,Z 969.227,A -85,B 0,C 180,E1 10944.272,E2 10944.272} C_VEL
LIN {X 0,Y 442.896,Z 988.262,A -85,B 0,C 180,E1 10942.973,E2 10942.973} C_VEL
LIN {X 0,Y 434.128,Z 1011.184,A -85,B 0,C 180,E1 10941.122,E2 10941.122} C_VEL
LIN {X 0,Y 426.073,Z 1030.341,A -85,B 0,C 180,E1 10939.277,E2 10939.277} C_VEL
LIN {X 0,Y 418.755,Z 1046.804,A -85,B 0,C 180,E1 10937.444,E2 10937.444} C_VEL
LIN {X 0,Y 409.913,Z 1065.874,A -85,B 0,C 180,E1 10934.977,E2 10934.977} C_VEL
LIN {X 0,Y 401.741,Z 1082.467,A -85,B 0,C 180,E1 10932.414,E2 10932.414} C_VEL
LIN {X 0,Y 394.989,Z 1095.939,A -85,B 0,C 180,E1 10930.015,E2 10930.015} C_VEL
LIN {X 0,Y 388.193,Z 1109.418,A -85,B 0,C 180,E1 10927.25,E2 10927.25} C_VEL
LIN {X 0,Y 380.728,Z 1124.273,A -85,B 0,C 180,E1 10923.641,E2 10923.641} C_VEL
LIN {X 0,Y 375.512,Z 1134.923,A -85,B 0,C 180,E1 10920.569,E2 10920.569} C_VEL
LIN {X 0,Y 371.133,Z 1144.295,A -85,B 0,C 180,E1 10917.432,E2 10917.432} C_VEL
LIN {X 0,Y 366.869,Z 1154.329,A -85,B 0,C 180,E1 10913.448,E2 10913.448} C_VEL
LIN {X 0,Y 363.899,Z 1162.123,A -85,B 0,C 180,E1 10909.586,E2 10909.586} C_VEL
LIN {X 0,Y 362.126,Z 1167.741,A -85,B 0,C 180,E1 10906.193,E2 10906.193} C_VEL
LIN {X 0,Y 360.949,Z 1172.446,A -85,B 0,C 180,E1 10902.641,E2 10902.641} C_VEL
LIN {X 0,Y 360.251,Z 1176.571,A -85,B 0,C 180,E1 10898.299,E2 10898.299} C_VEL
LIN {X 0,Y 360.023,Z 1178.628,A -85,B 0,C 180,E1 10894.78,E2 10894.78} C_VEL
LIN {X 0,Y 359.978,Z 1179.552,A -85,B 0,C 180,E1 10891.592,E2 10891.592} C_VEL
LIN {X 0,Y 359.984,Z 1179.587,A -85,B 0,C 180,E1 10888.568,E2 10888.568} C_VEL
LIN {X 0,Y 360.015,Z 1178.734,A -85,B 0,C 180,E1 10885.381,E2 10885.381} C_VEL
LIN {X 0,Y 360.19,Z 1176.964,A -85,B 0,C 180,E1 10882.183,E2 10882.183} C_VEL
LIN {X 0,Y 360.654,Z 1173.957,A -85,B 0,C 180,E1 10878.648,E2 10878.648} C_VEL
LIN {X 0,Y 361.897,Z 1168.624,A -85,B 0,C 180,E1 10874.291,E2 10874.291} C_VEL
LIN {X 0,Y 363.653,Z 1162.886,A -85,B 0,C 180,E1 10870.735,E2 10870.735} C_VEL
LIN {X 0,Y 365.722,Z 1157.168,A -85,B 0,C 180,E1 10867.79,E2 10867.79} C_VEL
LIN {X 0,Y 365.725,Z 1154.883,A -85,B 0,C 180,E1 10866.628,E2 10866.628} C_VEL
LIN {X 0,Y 362.683,Z 1148.686,A -85,B 0,C 180,E1 10863.462,E2 10863.462} C_VEL
LIN {X 0,Y 363.074,Z 1146.263,A -85,B 0,C 180,E1 10862.483,E2 10862.483} C_VEL
LIN {X 0,Y 368.047,Z 1135.988,A -85,B 0,C 180,E1 10858.924,E2 10858.924} C_VEL
LIN {X 0,Y 373.455,Z 1125.399,A -85,B 0,C 180,E1 10855.789,E2 10855.789} C_VEL
LIN {X 0,Y 380.81,Z 1111.47,A -85,B 0,C 180,E1 10852.282,E2 10852.282} C_VEL
LIN {X 0,Y 388.153,Z 1097.425,A -85,B 0,C 180,E1 10849.329,E2 10849.329} C_VEL
LIN {X 0,Y 395.096,Z 1084.072,A -85,B 0,C 180,E1 10846.899,E2 10846.899} C_VEL
LIN {X 0,Y 402.66,Z 1069.211,A -85,B 0,C 180,E1 10844.548,E2 10844.548} C_VEL
LIN {X 0,Y 412.743,Z 1048.465,A -85,B 0,C 180,E1 10841.775,E2 10841.775} C_VEL
LIN {X 0,Y 420.623,Z 1031.306,A -85,B 0,C 180,E1 10839.842,E2 10839.842} C_VEL
LIN {X 0,Y 428.303,Z 1013.608,A -85,B 0,C 180,E1 10838.12,E2 10838.12} C_VEL
LIN {X 0,Y 437.496,Z 990.584,A -85,B 0,C 180,E1 10836.219,E2 10836.219} C_VEL
LIN {X 0,Y 444.691,Z 970.66,A -85,B 0,C 180,E1 10834.846,E2 10834.846} C_VEL
LIN {X 0,Y 450.868,Z 951.879,A -85,B 0,C 180,E1 10833.734,E2 10833.734} C_VEL
LIN {X 0,Y 457.528,Z 929.305,A -85,B 0,C 180,E1 10832.599,E2 10832.599} C_VEL
LIN {X 0,Y 463.851,Z 903.955,A -85,B 0,C 180,E1 10831.57,E2 10831.57} C_VEL
LIN {X 0,Y 468.395,Z 882.318,A -85,B 0,C 180,E1 10830.862,E2 10830.862} C_VEL
LIN {X 0,Y 472.346,Z 859.724,A -85,B 0,C 180,E1 10830.277,E2 10830.277} C_VEL
LIN {X 0,Y 475.893,Z 831.342,A -85,B 0,C 180,E1 10829.716,E2 10829.716} C_VEL
LIN {X 0,Y 481.851,Z 747.942,A -85,B 0,C 180,E1 10828.418,E2 10828.418} C_VEL
LIN {X 0,Y 497.118,Z 534.836,A -85,B 0,C 180,E1 10825.155,E2 10825.155} C_VEL
LIN {X 0,Y 490.77,Z 523.461,A -85,B 0,C 180,E1 10822.901,E2 10822.901} C_VEL
LIN {X 0,Y 485.069,Z 513.522,A -85,B 0,C 180,E1 10820.608,E2 10820.608} C_VEL
LIN {X 0,Y 479.752,Z 504.782,A -85,B 0,C 180,E1 10818.155,E2 10818.155} C_VEL
LIN {X 0,Y 475.65,Z 497.949,A -85,B 0,C 180,E1 10815.922,E2 10815.922} C_VEL
LIN {X 0,Y 472.209,Z 492.563,A -85,B 0,C 180,E1 10813.719,E2 10813.719} C_VEL
LIN {X 0,Y 469.45,Z 488.121,A -85,B 0,C 180,E1 10811.549,E2 10811.549} C_VEL
LIN {X 0,Y 467.071,Z 484.128,A -85,B 0,C 180,E1 10809.115,E2 10809.115} C_VEL
LIN {X 0,Y 464.571,Z 479.605,A -85,B 0,C 180,E1 10804.568,E2 10804.568} C_VEL
LIN {X 0,Y 464.426,Z 479.084,A -85,B 0,C 180,E1 10800.37,E2 10800.37} C_VEL
LIN {X 0,Y 466.234,Z 480.465,A -85,B 0,C 180,E1 10796.557,E2 10796.557} C_VEL
LIN {X 0,Y 470.407,Z 486.016,A -85,B 0,C 180,E1 10792.181,E2 10792.181} C_VEL
LIN {X 0,Y 474.177,Z 491.166,A -85,B 0,C 180,E1 10789.49,E2 10789.49} C_VEL
LIN {X 0,Y 478.137,Z 496.746,A -85,B 0,C 180,E1 10787.193,E2 10787.193} C_VEL
LIN {X 0,Y 481.86,Z 502.099,A -85,B 0,C 180,E1 10785.335,E2 10785.335} C_VEL
LIN {X 0,Y 487.084,Z 509.827,A -85,B 0,C 180,E1 10783.052,E2 10783.052} C_VEL
LIN {X 0,Y 494.776,Z 521.75,A -85,B 0,C 180,E1 10780.153,E2 10780.153} C_VEL
LIN {X 0,Y 499.607,Z 529.935,A -85,B 0,C 180,E1 10778.518,E2 10778.518} C_VEL
LIN {X 0,Y 483.207,Z 748.552,A -85,B 0,C 180,E1 10775.042,E2 10775.042} C_VEL
LIN {X 0,Y 477.186,Z 828.329,A -85,B 0,C 180,E1 10773.746,E2 10773.746} C_VEL
LIN {X 0,Y 473.572,Z 856.906,A -85,B 0,C 180,E1 10773.173,E2 10773.173} C_VEL
LIN {X 0,Y 469.363,Z 880.949,A -85,B 0,C 180,E1 10772.539,E2 10772.539} C_VEL
LIN {X 0,Y 464.963,Z 902.039,A -85,B 0,C 180,E1 10771.845,E2 10771.845} C_VEL
LIN {X 0,Y 459.876,Z 923.026,A -85,B 0,C 180,E1 10771.019,E2 10771.019} C_VEL
LIN {X 0,Y 452.72,Z 948.826,A -85,B 0,C 180,E1 10769.788,E2 10769.788} C_VEL
LIN {X 0,Y 445.456,Z 971.572,A -85,B 0,C 180,E1 10768.466,E2 10768.466} C_VEL
LIN {X 0,Y 438.583,Z 991.181,A -85,B 0,C 180,E1 10767.139,E2 10767.139} C_VEL
LIN {X 0,Y 430.693,Z 1012.058,A -85,B 0,C 180,E1 10765.496,E2 10765.496} C_VEL
LIN {X 0,Y 421.04,Z 1035.496,A -85,B 0,C 180,E1 10763.305,E2 10763.305} C_VEL
LIN {X 0,Y 413.095,Z 1053.624,A -85,B 0,C 180,E1 10761.315,E2 10761.315} C_VEL
LIN {X 0,Y 405.388,Z 1070.517,A -85,B 0,C 180,E1 10759.184,E2 10759.184} C_VEL
LIN {X 0,Y 396.365,Z 1089.711,A -85,B 0,C 180,E1 10756.385,E2 10756.385} C_VEL
LIN {X 0,Y 387.944,Z 1107.036,A -85,B 0,C 180,E1 10753.378,E2 10753.378} C_VEL
LIN {X 0,Y 381.504,Z 1120.292,A -85,B 0,C 180,E1 10750.737,E2 10750.737} C_VEL
LIN {X 0,Y 375.31,Z 1133.249,A -85,B 0,C 180,E1 10747.788,E2 10747.788} C_VEL
LIN {X 0,Y 368.362,Z 1148.223,A -85,B 0,C 180,E1 10743.81,E2 10743.81} C_VEL
LIN {X 0,Y 363.421,Z 1159.533,A -85,B 0,C 180,E1 10740.23,E2 10740.23} C_VEL
LIN {X 0,Y 359.731,Z 1168.762,A -85,B 0,C 180,E1 10736.844,E2 10736.844} C_VEL
LIN {X 0,Y 356.779,Z 1177.097,A -85,B 0,C 180,E1 10733.275,E2 10733.275} C_VEL
LIN {X 0,Y 354.221,Z 1185.769,A -85,B 0,C 180,E1 10728.771,E2 10728.771} C_VEL
LIN {X 0,Y 352.934,Z 1191.557,A -85,B 0,C 180,E1 10724.94,E2 10724.94} C_VEL
LIN {X 0,Y 352.279,Z 1195.695,A -85,B 0,C 180,E1 10721.46,E2 10721.46} C_VEL
LIN {X 0,Y 352.04,Z 1198.502,A -85,B 0,C 180,E1 10718.328,E2 10718.328} C_VEL
LIN {X 0,Y 351.96,Z 1200.495,A -85,B 0,C 180,E1 10715.052,E2 10715.052} C_VEL
LIN {X 0,Y 351.954,Z 1201.49,A -85,B 0,C 180,E1 10711.953,E2 10711.953} C_VEL
LIN {X 0,Y 351.957,Z 1201.609,A -85,B 0,C 180,E1 10708.86,E2 10708.86} C_VEL
LIN {X 0,Y 351.952,Z 1200.779,A -85,B 0,C 180,E1 10705.6,E2 10705.6} C_VEL
LIN {X 0,Y 352.014,Z 1198.976,A -85,B 0,C 180,E1 10702.328,E2 10702.328} C_VEL
LIN {X 0,Y 352.23,Z 1196.193,A -85,B 0,C 180,E1 10699.036,E2 10699.036} C_VEL
LIN {X 0,Y 352.776,Z 1192.416,A -85,B 0,C 180,E1 10695.724,E2 10695.724} C_VEL
LIN {X 0,Y 353.747,Z 1187.623,A -85,B 0,C 180,E1 10692.395,E2 10692.395} C_VEL
LIN {X 0,Y 355.31,Z 1181.786,A -85,B 0,C 180,E1 10689.06,E2 10689.06} C_VEL
LIN {X 0,Y 357.645,Z 1174.501,A -85,B 0,C 180,E1 10685.558,E2 10685.558} C_VEL
LIN {X 0,Y 361.703,Z 1163.794,A -85,B 0,C 180,E1 10681.249,E2 10681.249} C_VEL
LIN {X 0,Y 366.467,Z 1152.413,A -85,B 0,C 180,E1 10677.469,E2 10677.469} C_VEL
LIN {X 0,Y 371.513,Z 1141.246,A -85,B 0,C 180,E1 10674.265,E2 10674.265} C_VEL
LIN {X 0,Y 377.475,Z 1128.621,A -85,B 0,C 180,E1 10671.113,E2 10671.113} C_VEL
LIN {X 0,Y 386.094,Z 1110.823,A -85,B 0,C 180,E1 10667.349,E2 10667.349} C_VEL
LIN {X 0,Y 392.972,Z 1096.579,A -85,B 0,C 180,E1 10664.774,E2 10664.774} C_VEL
LIN {X 0,Y 399.968,Z 1081.961,A -85,B 0,C 180,E1 10662.453,E2 10662.453} C_VEL
LIN {X 0,Y 407.392,Z 1066.113,A -85,B 0,C 180,E1 10660.244,E2 10660.244} C_VEL
LIN {X 0,Y 416.76,Z 1045.423,A -85,B 0,C 180,E1 10657.754,E2 10657.754} C_VEL
LIN {X 0,Y 425.38,Z 1025.015,A -85,B 0,C 180,E1 10655.685,E2 10655.685} C_VEL
LIN {X 0,Y 432.43,Z 1007.357,A -85,B 0,C 180,E1 10654.129,E2 10654.129} C_VEL
LIN {X 0,Y 439.497,Z 988.437,A -85,B 0,C 180,E1 10652.672,E2 10652.672} C_VEL
LIN {X 0,Y 447.793,Z 964.433,A -85,B 0,C 180,E1 10651.094,E2 10651.094} C_VEL
LIN {X 0,Y 455.075,Z 940.258,A -85,B 0,C 180,E1 10649.786,E2 10649.786} C_VEL
LIN {X 0,Y 460.617,Z 919.703,A -85,B 0,C 180,E1 10648.849,E2 10648.849} C_VEL
LIN {X 0,Y 465.611,Z 898.677,A -85,B 0,C 180,E1 10648.042,E2 10648.042} C_VEL
LIN {X 0,Y 470.961,Z 872.194,A -85,B 0,C 180,E1 10647.215,E2 10647.215} C_VEL
LIN {X 0,Y 474.979,Z 846.084,A -85,B 0,C 180,E1 10646.601,E2 10646.601} C_VEL
LIN {X 0,Y 477.511,Z 823.58,A -85,B 0,C 180,E1 10646.179,E2 10646.179} C_VEL
LIN {X 0,Y 493.232,Z 612.153,A -85,B 0,C 180,E1 10642.792,E2 10642.792} C_VEL
LIN {X 0,Y 499.431,Z 529.548,A -85,B 0,C 180,E1 10641.462,E2 10641.462} C_VEL
LIN {X 0,Y 491.938,Z 517.389,A -85,B 0,C 180,E1 10638.886,E2 10638.886} C_VEL
LIN {X 0,Y 485.162,Z 507.047,A -85,B 0,C 180,E1 10636.216,E2 10636.216} C_VEL
LIN {X 0,Y 479.668,Z 498.933,A -85,B 0,C 180,E1 10633.686,E2 10633.686} C_VEL
LIN {X 0,Y 476.138,Z 494.073,A -85,B 0,C 180,E1 10631.815,E2 10631.815} C_VEL
LIN {X 0,Y 472.975,Z 489.594,A -85,B 0,C 180,E1 10629.86,E2 10629.86} C_VEL
LIN {X 0,Y 469.612,Z 485.047,A -85,B 0,C 180,E1 10627.34,E2 10627.34} C_VEL
LIN {X 0,Y 465.824,Z 480.04,A -85,B 0,C 180,E1 10623.199,E2 10623.199} C_VEL
LIN {X 0,Y 463.997,Z 478.808,A -85,B 0,C 180,E1 10618.765,E2 10618.765} C_VEL
LIN {X 0,Y 464.527,Z 479.682,A -85,B 0,C 180,E1 10614.689,E2 10614.689} C_VEL
LIN {X 0,Y 467.518,Z 484.981,A -85,B 0,C 180,E1 10610.024,E2 10610.024} C_VEL
LIN {X 0,Y 470.435,Z 489.865,A -85,B 0,C 180,E1 10607.354,E2 10607.354} C_VEL
LIN {X 0,Y 473.474,Z 494.699,A -85,B 0,C 180,E1 10605.195,E2 10605.195} C_VEL
LIN {X 0,Y 478.117,Z 502.098,A -85,B 0,C 180,E1 10602.505,E2 10602.505} C_VEL
LIN {X 0,Y 483.406,Z 510.9,A -85,B 0,C 180,E1 10599.95,E2 10599.95} C_VEL
LIN {X 0,Y 489.83,Z 521.909,A -85,B 0,C 180,E1 10597.306,E2 10597.306} C_VEL
LIN {X 0,Y 496.487,Z 533.84,A -85,B 0,C 180,E1 10594.917,E2 10594.917} C_VEL
LIN {X 0,Y 496.969,Z 535.033,A -85,B 0,C 180,E1 10594.744,E2 10594.744} C_VEL
LIN {X 0,Y 481.102,Z 756.951,A -85,B 0,C 180,E1 10591.347,E2 10591.347} C_VEL
LIN {X 0,Y 475.728,Z 831.771,A -85,B 0,C 180,E1 10590.179,E2 10590.179} C_VEL
LIN {X 0,Y 472.09,Z 860.55,A -85,B 0,C 180,E1 10589.604,E2 10589.604} C_VEL
LIN {X 0,Y 468.236,Z 882.506,A -85,B 0,C 180,E1 10589.035,E2 10589.035} C_VEL
LIN {X 0,Y 463.583,Z 904.625,A -85,B 0,C 180,E1 10588.307,E2 10588.307} C_VEL
LIN {X 0,Y 456.779,Z 931.481,A -85,B 0,C 180,E1 10587.2,E2 10587.2} C_VEL
LIN {X 0,Y 450.462,Z 952.813,A -85,B 0,C 180,E1 10586.115,E2 10586.115} C_VEL
LIN {X 0,Y 444.307,Z 971.485,A -85,B 0,C 180,E1 10585,E2 10585} C_VEL
LIN {X 0,Y 436.268,Z 993.699,A -85,B 0,C 180,E1 10583.447,E2 10583.447} C_VEL
LIN {X 0,Y 427.676,Z 1014.853,A -85,B 0,C 180,E1 10581.663,E2 10581.663} C_VEL
LIN {X 0,Y 420.299,Z 1031.84,A -85,B 0,C 180,E1 10579.999,E2 10579.999} C_VEL
LIN {X 0,Y 412.271,Z 1049.332,A -85,B 0,C 180,E1 10578.018,E2 10578.018} C_VEL
LIN {X 0,Y 402.552,Z 1069.292,A -85,B 0,C 180,E1 10575.337,E2 10575.337} C_VEL
LIN {X 0,Y 394.851,Z 1084.429,A -85,B 0,C 180,E1 10572.937,E2 10572.937} C_VEL
LIN {X 0,Y 387.546,Z 1098.497,A -85,B 0,C 180,E1 10570.36,E2 10570.36} C_VEL
LIN {X 0,Y 378.912,Z 1114.896,A -85,B 0,C 180,E1 10566.799,E2 10566.799} C_VEL
LIN {X 0,Y 372.723,Z 1126.747,A -85,B 0,C 180,E1 10563.732,E2 10563.732} C_VEL
LIN {X 0,Y 367.189,Z 1137.694,A -85,B 0,C 180,E1 10560.431,E2 10560.431} C_VEL
LIN {X 0,Y 361.69,Z 1149.189,A -85,B 0,C 180,E1 10556.252,E2 10556.252} C_VEL
LIN {X 0,Y 358.29,Z 1156.972,A -85,B 0,C 180,E1 10552.825,E2 10552.825} C_VEL
LIN {X 0,Y 355.77,Z 1163.547,A -85,B 0,C 180,E1 10549.368,E2 10549.368} C_VEL
LIN {X 0,Y 353.706,Z 1170.138,A -85,B 0,C 180,E1 10545.075,E2 10545.075} C_VEL
LIN {X 0,Y 352.629,Z 1174.568,A -85,B 0,C 180,E1 10541.117,E2 10541.117} C_VEL
LIN {X 0,Y 352.204,Z 1177.288,A -85,B 0,C 180,E1 10537.778,E2 10537.778} C_VEL
LIN {X 0,Y 352.021,Z 1179.053,A -85,B 0,C 180,E1 10534.442,E2 10534.442} C_VEL
LIN {X 0,Y 351.985,Z 1179.863,A -85,B 0,C 180,E1 10531.14,E2 10531.14} C_VEL
LIN {X 0,Y 351.992,Z 1179.727,A -85,B 0,C 180,E1 10527.721,E2 10527.721} C_VEL
LIN {X 0,Y 352.101,Z 1178.295,A -85,B 0,C 180,E1 10523.642,E2 10523.642} C_VEL
LIN {X 0,Y 352.484,Z 1175.424,A -85,B 0,C 180,E1 10519.706,E2 10519.706} C_VEL
LIN {X 0,Y 353.244,Z 1171.837,A -85,B 0,C 180,E1 10516.246,E2 10516.246} C_VEL
LIN {X 0,Y 354.564,Z 1167.175,A -85,B 0,C 180,E1 10512.777,E2 10512.777} C_VEL
LIN {X 0,Y 357.058,Z 1160.232,A -85,B 0,C 180,E1 10508.652,E2 10508.652} C_VEL
LIN {X 0,Y 360.703,Z 1151.379,A -85,B 0,C 180,E1 10504.554,E2 10504.554} C_VEL
LIN {X 0,Y 363.074,Z 1146.263,A -85,B 0,C 180,E1 10502.483,E2 10502.483} C_VEL
LIN {X 0,Y 363.503,Z 1143.428,A -85,B 0,C 180,E1 10501.349,E2 10501.349} C_VEL
LIN {X 0,Y 361.783,Z 1135.966,A -85,B 0,C 180,E1 10498.215,E2 10498.215} C_VEL
LIN {X 0,Y 362.617,Z 1133.2,A -85,B 0,C 180,E1 10497.261,E2 10497.261} C_VEL
LIN {X 0,Y 370.153,Z 1119.242,A -85,B 0,C 180,E1 10493.347,E2 10493.347} C_VEL
LIN {X 0,Y 376.859,Z 1106.979,A -85,B 0,C 180,E1 10490.45,E2 10490.45} C_VEL
LIN {X 0,Y 384.393,Z 1093.205,A -85,B 0,C 180,E1 10487.647,E2 10487.647} C_VEL
LIN {X 0,Y 394.12,Z 1074.963,A -85,B 0,C 180,E1 10484.53,E2 10484.53} C_VEL
LIN {X 0,Y 402.047,Z 1059.482,A -85,B 0,C 180,E1 10482.291,E2 10482.291} C_VEL
LIN {X 0,Y 410.052,Z 1043.191,A -85,B 0,C 180,E1 10480.251,E2 10480.251} C_VEL
LIN {X 0,Y 419.924,Z 1021.868,A -85,B 0,C 180,E1 10477.988,E2 10477.988} C_VEL
LIN {X 0,Y 427.993,Z 1002.87,A -85,B 0,C 180,E1 10476.295,E2 10476.295} C_VEL
LIN {X 0,Y 435.182,Z 984.611,A -85,B 0,C 180,E1 10474.891,E2 10474.891} C_VEL
LIN {X 0,Y 443.279,Z 962.232,A -85,B 0,C 180,E1 10473.428,E2 10473.428} C_VEL
LIN {X 0,Y 450.768,Z 938.376,A -85,B 0,C 180,E1 10472.149,E2 10472.149} C_VEL
LIN {X 0,Y 456.235,Z 918.755,A -85,B 0,C 180,E1 10471.272,E2 10471.272} C_VEL
LIN {X 0,Y 460.919,Z 899.555,A -85,B 0,C 180,E1 10470.547,E2 10470.547} C_VEL
LIN {X 0,Y 465.926,Z 875.413,A -85,B 0,C 180,E1 10469.798,E2 10469.798} C_VEL
LIN {X 0,Y 470.118,Z 848.943,A -85,B 0,C 180,E1 10469.182,E2 10469.182} C_VEL
LIN {X 0,Y 472.613,Z 826.704,A -85,B 0,C 180,E1 10468.778,E2 10468.778} C_VEL
LIN {X 0,Y 489.376,Z 596.402,A -85,B 0,C 180,E1 10465.238,E2 10465.238} C_VEL
LIN {X 0,Y 493.6,Z 539.443,A -85,B 0,C 180,E1 10464.345,E2 10464.345} C_VEL
LIN {X 0,Y 486.265,Z 526.057,A -85,B 0,C 180,E1 10461.565,E2 10461.565} C_VEL
LIN {X 0,Y 479.783,Z 514.934,A -85,B 0,C 180,E1 10458.689,E2 10458.689} C_VEL
LIN {X 0,Y 474.968,Z 506.888,A -85,B 0,C 180,E1 10456.134,E2 10456.134} C_VEL
LIN {X 0,Y 470.982,Z 500.378,A -85,B 0,C 180,E1 10453.568,E2 10453.568} C_VEL
LIN {X 0,Y 468.204,Z 495.83,A -85,B 0,C 180,E1 10451.331,E2 10451.331} C_VEL
LIN {X 0,Y 465.999,Z 492.011,A -85,B 0,C 180,E1 10449.012,E2 10449.012} C_VEL
LIN {X 0,Y 463.6,Z 487.554,A -85,B 0,C 180,E1 10444.577,E2 10444.577} C_VEL
LIN {X 0,Y 463.451,Z 487.025,A -85,B 0,C 180,E1 10440.371,E2 10440.371} C_VEL
LIN {X 0,Y 465.241,Z 488.488,A -85,B 0,C 180,E1 10436.55,E2 10436.55} C_VEL
LIN {X 0,Y 469.19,Z 493.819,A -85,B 0,C 180,E1 10432.346,E2 10432.346} C_VEL
LIN {X 0,Y 472.802,Z 498.85,A -85,B 0,C 180,E1 10429.706,E2 10429.706} C_VEL
LIN {X 0,Y 476.689,Z 504.44,A -85,B 0,C 180,E1 10427.4,E2 10427.4} C_VEL
LIN {X 0,Y 480.478,Z 509.989,A -85,B 0,C 180,E1 10425.477,E2 10425.477} C_VEL
LIN {X 0,Y 486.119,Z 518.584,A -85,B 0,C 180,E1 10422.987,E2 10422.987} C_VEL
LIN {X 0,Y 493.02,Z 529.537,A -85,B 0,C 180,E1 10420.357,E2 10420.357} C_VEL
LIN {X 0,Y 496.059,Z 534.917,A -85,B 0,C 180,E1 10419.289,E2 10419.289} C_VEL
LIN {X 0,Y 479.292,Z 753.133,A -85,B 0,C 180,E1 10415.825,E2 10415.825} C_VEL
LIN {X 0,Y 473.436,Z 828.532,A -85,B 0,C 180,E1 10414.599,E2 10414.599} C_VEL
LIN {X 0,Y 469.688,Z 857.4,A -85,B 0,C 180,E1 10414.021,E2 10414.021} C_VEL
LIN {X 0,Y 465.46,Z 881.037,A -85,B 0,C 180,E1 10413.401,E2 10413.401} C_VEL
LIN {X 0,Y 460.987,Z 902.018,A -85,B 0,C 180,E1 10412.715,E2 10412.715} C_VEL
LIN {X 0,Y 455.728,Z 923.248,A -85,B 0,C 180,E1 10411.883,E2 10411.883} C_VEL
LIN {X 0,Y 448.299,Z 949.327,A -85,B 0,C 180,E1 10410.64,E2 10410.64} C_VEL
LIN {X 0,Y 441.139,Z 971.217,A -85,B 0,C 180,E1 10409.373,E2 10409.373} C_VEL
LIN {X 0,Y 434.123,Z 990.765,A -85,B 0,C 180,E1 10408.056,E2 10408.056} C_VEL
LIN {X 0,Y 426.644,Z 1010.096,A -85,B 0,C 180,E1 10406.544,E2 10406.544} C_VEL
LIN {X 0,Y 416.862,Z 1033.443,A -85,B 0,C 180,E1 10404.401,E2 10404.401} C_VEL
LIN {X 0,Y 408.171,Z 1052.698,A -85,B 0,C 180,E1 10402.301,E2 10402.301} C_VEL
LIN {X 0,Y 400.268,Z 1069.492,A -85,B 0,C 180,E1 10400.187,E2 10400.187} C_VEL
LIN {X 0,Y 391.268,Z 1088.012,A -85,B 0,C 180,E1 10397.498,E2 10397.498} C_VEL
LIN {X 0,Y 382.342,Z 1105.716,A -85,B 0,C 180,E1 10394.443,E2 10394.443} C_VEL
LIN {X 0,Y 375.482,Z 1119.265,A -85,B 0,C 180,E1 10391.738,E2 10391.738} C_VEL
LIN {X 0,Y 369.282,Z 1131.64,A -85,B 0,C 180,E1 10388.915,E2 10388.915} C_VEL
LIN {X 0,Y 363.001,Z 1144.539,A -85,B 0,C 180,E1 10385.534,E2 10385.534} C_VEL
LIN {X 0,Y 356.545,Z 1158.425,A -85,B 0,C 180,E1 10381.202,E2 10381.202} C_VEL
LIN {X 0,Y 352.523,Z 1167.838,A -85,B 0,C 180,E1 10377.72,E2 10377.72} C_VEL
LIN {X 0,Y 349.507,Z 1175.721,A -85,B 0,C 180,E1 10374.328,E2 10374.328} C_VEL
LIN {X 0,Y 347.182,Z 1182.799,A -85,B 0,C 180,E1 10370.746,E2 10370.746} C_VEL
LIN {X 0,Y 345.313,Z 1189.995,A -85,B 0,C 180,E1 10366.312,E2 10366.312} C_VEL
LIN {X 0,Y 344.36,Z 1195.104,A -85,B 0,C 180,E1 10362.067,E2 10362.067} C_VEL
LIN {X 0,Y 344.056,Z 1198.131,A -85,B 0,C 180,E1 10358.691,E2 10358.691} C_VEL
LIN {X 0,Y 343.965,Z 1200.174,A -85,B 0,C 180,E1 10355.337,E2 10355.337} C_VEL
LIN {X 0,Y 343.958,Z 1201.219,A -85,B 0,C 180,E1 10352.165,E2 10352.165} C_VEL
LIN {X 0,Y 343.961,Z 1201.362,A -85,B 0,C 180,E1 10348.834,E2 10348.834} C_VEL
LIN {X 0,Y 343.957,Z 1200.53,A -85,B 0,C 180,E1 10345.498,E2 10345.498} C_VEL
LIN {X 0,Y 344.019,Z 1198.725,A -85,B 0,C 180,E1 10342.148,E2 10342.148} C_VEL
LIN {X 0,Y 344.253,Z 1195.937,A -85,B 0,C 180,E1 10338.778,E2 10338.778} C_VEL
LIN {X 0,Y 344.849,Z 1192.157,A -85,B 0,C 180,E1 10335.389,E2 10335.389} C_VEL
LIN {X 0,Y 345.899,Z 1187.359,A -85,B 0,C 180,E1 10331.983,E2 10331.983} C_VEL
LIN {X 0,Y 347.564,Z 1181.517,A -85,B 0,C 180,E1 10328.57,E2 10328.57} C_VEL
LIN {X 0,Y 350.059,Z 1174.228,A -85,B 0,C 180,E1 10324.992,E2 10324.992} C_VEL
LIN {X 0,Y 354.348,Z 1163.509,A -85,B 0,C 180,E1 10320.594,E2 10320.594} C_VEL
LIN {X 0,Y 359.361,Z 1152.172,A -85,B 0,C 180,E1 10316.761,E2 10316.761} C_VEL
LIN {X 0,Y 364.668,Z 1140.949,A -85,B 0,C 180,E1 10313.488,E2 10313.488} C_VEL
LIN {X 0,Y 371.27,Z 1127.661,A -85,B 0,C 180,E1 10310.135,E2 10310.135} C_VEL
LIN {X 0,Y 379.67,Z 1110.995,A -85,B 0,C 180,E1 10306.579,E2 10306.579} C_VEL
LIN {X 0,Y 387.063,Z 1096.252,A -85,B 0,C 180,E1 10303.885,E2 10303.885} C_VEL
LIN {X 0,Y 394.488,Z 1081.284,A -85,B 0,C 180,E1 10301.497,E2 10301.497} C_VEL
LIN {X 0,Y 402.51,Z 1064.724,A -85,B 0,C 180,E1 10299.191,E2 10299.191} C_VEL
LIN {X 0,Y 412.986,Z 1041.993,A -85,B 0,C 180,E1 10296.505,E2 10296.505} C_VEL
LIN {X 0,Y 420.818,Z 1023.995,A -85,B 0,C 180,E1 10294.703,E2 10294.703} C_VEL
LIN {X 0,Y 427.821,Z 1006.924,A -85,B 0,C 180,E1 10293.207,E2 10293.207} C_VEL
LIN {X 0,Y 435.08,Z 987.974,A -85,B 0,C 180,E1 10291.754,E2 10291.754} C_VEL
LIN {X 0,Y 443.611,Z 963.795,A -85,B 0,C 180,E1 10290.175,E2 10290.175} C_VEL
LIN {X 0,Y 451.043,Z 939.648,A -85,B 0,C 180,E1 10288.879,E2 10288.879} C_VEL
LIN {X 0,Y 456.601,Z 919.46,A -85,B 0,C 180,E1 10287.966,E2 10287.966} C_VEL
LIN {X 0,Y 461.821,Z 897.891,A -85,B 0,C 180,E1 10287.146,E2 10287.146} C_VEL
LIN {X 0,Y 467.368,Z 870.568,A -85,B 0,C 180,E1 10286.311,E2 10286.311} C_VEL
LIN {X 0,Y 471.234,Z 845.859,A -85,B 0,C 180,E1 10285.738,E2 10285.738} C_VEL
LIN {X 0,Y 473.806,Z 823.356,A -85,B 0,C 180,E1 10285.319,E2 10285.319} C_VEL
LIN {X 0,Y 490.095,Z 609.804,A -85,B 0,C 180,E1 10281.902,E2 10281.902} C_VEL
LIN {X 0,Y 495.893,Z 534.519,A -85,B 0,C 180,E1 10280.693,E2 10280.693} C_VEL
LIN {X 0,Y 489.546,Z 524.079,A -85,B 0,C 180,E1 10278.426,E2 10278.426} C_VEL
LIN {X 0,Y 483.211,Z 514.198,A -85,B 0,C 180,E1 10275.851,E2 10275.851} C_VEL
LIN {X 0,Y 477.847,Z 506.166,A -85,B 0,C 180,E1 10273.307,E2 10273.307} C_VEL
LIN {X 0,Y 474.621,Z 501.622,A -85,B 0,C 180,E1 10271.545,E2 10271.545} C_VEL
LIN {X 0,Y 471.531,Z 497.186,A -85,B 0,C 180,E1 10269.582,E2 10269.582} C_VEL
LIN {X 0,Y 468.337,Z 492.785,A -85,B 0,C 180,E1 10267.113,E2 10267.113} C_VEL
LIN {X 0,Y 464.759,Z 487.937,A -85,B 0,C 180,E1 10263.083,E2 10263.083} C_VEL
LIN {X 0,Y 463.022,Z 486.749,A -85,B 0,C 180,E1 10258.763,E2 10258.763} C_VEL
LIN {X 0,Y 463.511,Z 487.57,A -85,B 0,C 180,E1 10254.802,E2 10254.802} C_VEL
LIN {X 0,Y 466.375,Z 492.793,A -85,B 0,C 180,E1 10250.186,E2 10250.186} C_VEL
LIN {X 0,Y 469.235,Z 497.704,A -85,B 0,C 180,E1 10247.509,E2 10247.509} C_VEL
LIN {X 0,Y 472.045,Z 502.254,A -85,B 0,C 180,E1 10245.463,E2 10245.463} C_VEL
LIN {X 0,Y 476.585,Z 509.678,A -85,B 0,C 180,E1 10242.762,E2 10242.762} C_VEL
LIN {X 0,Y 481.653,Z 518.285,A -85,B 0,C 180,E1 10240.253,E2 10240.253} C_VEL
LIN {X 0,Y 487.812,Z 529.075,A -85,B 0,C 180,E1 10237.652,E2 10237.652} C_VEL
LIN {X 0,Y 493.518,Z 539.57,A -85,B 0,C 180,E1 10235.532,E2 10235.532} C_VEL
LIN {X 0,Y 477.235,Z 761.363,A -85,B 0,C 180,E1 10232.14,E2 10232.14} C_VEL
LIN {X 0,Y 472.004,Z 831.987,A -85,B 0,C 180,E1 10231.036,E2 10231.036} C_VEL
LIN {X 0,Y 468.28,Z 860.7,A -85,B 0,C 180,E1 10230.464,E2 10230.464} C_VEL
LIN {X 0,Y 464.314,Z 882.792,A -85,B 0,C 180,E1 10229.894,E2 10229.894} C_VEL
LIN {X 0,Y 459.615,Z 904.648,A -85,B 0,C 180,E1 10229.179,E2 10229.179} C_VEL
LIN {X 0,Y 452.828,Z 930.944,A -85,B 0,C 180,E1 10228.104,E2 10228.104} C_VEL
LIN {X 0,Y 446.682,Z 951.35,A -85,B 0,C 180,E1 10227.079,E2 10227.079} C_VEL
LIN {X 0,Y 440.355,Z 970.188,A -85,B 0,C 180,E1 10225.974,E2 10225.974} C_VEL
LIN {X 0,Y 432.98,Z 990.154,A -85,B 0,C 180,E1 10224.606,E2 10224.606} C_VEL
LIN {X 0,Y 423.545,Z 1013.265,A -85,B 0,C 180,E1 10222.709,E2 10222.709} C_VEL
LIN {X 0,Y 415.651,Z 1031.005,A -85,B 0,C 180,E1 10220.987,E2 10220.987} C_VEL
LIN {X 0,Y 407.617,Z 1048.044,A -85,B 0,C 180,E1 10219.071,E2 10219.071} C_VEL
LIN {X 0,Y 397.894,Z 1067.586,A -85,B 0,C 180,E1 10216.484,E2 10216.484} C_VEL
LIN {X 0,Y 389.302,Z 1083.909,A -85,B 0,C 180,E1 10213.905,E2 10213.905} C_VEL
LIN {X 0,Y 382.101,Z 1097.292,A -85,B 0,C 180,E1 10211.457,E2 10211.457} C_VEL
LIN {X 0,Y 373.751,Z 1112.709,A -85,B 0,C 180,E1 10208.169,E2 10208.169} C_VEL
LIN {X 0,Y 366.475,Z 1125.913,A -85,B 0,C 180,E1 10204.767,E2 10204.767} C_VEL
LIN {X 0,Y 361.106,Z 1135.974,A -85,B 0,C 180,E1 10201.742,E2 10201.742} C_VEL
LIN {X 0,Y 355.917,Z 1146.169,A -85,B 0,C 180,E1 10198.162,E2 10198.162} C_VEL
LIN {X 0,Y 351.174,Z 1156.215,A -85,B 0,C 180,E1 10193.848,E2 10193.848} C_VEL
LIN {X 0,Y 348.367,Z 1162.935,A -85,B 0,C 180,E1 10190.322,E2 10190.322} C_VEL
LIN {X 0,Y 346.397,Z 1168.5,A -85,B 0,C 180,E1 10186.778,E2 10186.778} C_VEL
LIN {X 0,Y 344.95,Z 1173.744,A -85,B 0,C 180,E1 10182.556,E2 10182.556} C_VEL
LIN {X 0,Y 344.27,Z 1177.287,A -85,B 0,C 180,E1 10178.35,E2 10178.35} C_VEL
LIN {X 0,Y 344.035,Z 1179.189,A -85,B 0,C 180,E1 10174.835,E2 10174.835} C_VEL
LIN {X 0,Y 343.986,Z 1180.046,A -85,B 0,C 180,E1 10171.666,E2 10171.666} C_VEL
LIN {X 0,Y 343.992,Z 1180.081,A -85,B 0,C 180,E1 10168.501,E2 10168.501} C_VEL
LIN {X 0,Y 344.026,Z 1179.294,A -85,B 0,C 180,E1 10165.333,E2 10165.333} C_VEL
LIN {X 0,Y 344.219,Z 1177.57,A -85,B 0,C 180,E1 10161.986,E2 10161.986} C_VEL
LIN {X 0,Y 344.709,Z 1174.763,A -85,B 0,C 180,E1 10158.455,E2 10158.455} C_VEL
LIN {X 0,Y 346.005,Z 1169.867,A -85,B 0,C 180,E1 10154.066,E2 10154.066} C_VEL
LIN {X 0,Y 348.093,Z 1163.694,A -85,B 0,C 180,E1 10150.013,E2 10150.013} C_VEL
LIN {X 0,Y 350.794,Z 1157.102,A -85,B 0,C 180,E1 10146.482,E2 10146.482} C_VEL
LIN {X 0,Y 354.801,Z 1148.515,A -85,B 0,C 180,E1 10142.655,E2 10142.655} C_VEL
LIN {X 0,Y 360.475,Z 1137.258,A -85,B 0,C 180,E1 10138.569,E2 10138.569} C_VEL
LIN {X 0,Y 362.617,Z 1133.2,A -85,B 0,C 180,E1 10137.261,E2 10137.261} C_VEL
LIN {X 0,Y 363.562,Z 1129.962,A -85,B 0,C 180,E1 10136.157,E2 10136.157} C_VEL
LIN {X 0,Y 363.172,Z 1121.312,A -85,B 0,C 180,E1 10133.1,E2 10133.1} C_VEL
LIN {X 0,Y 364.364,Z 1118.068,A -85,B 0,C 180,E1 10132.2,E2 10132.2} C_VEL
LIN {X 0,Y 371.311,Z 1105.899,A -85,B 0,C 180,E1 10129.333,E2 10129.333} C_VEL
LIN {X 0,Y 380.552,Z 1089.636,A -85,B 0,C 180,E1 10126.081,E2 10126.081} C_VEL
LIN {X 0,Y 389.364,Z 1073.46,A -85,B 0,C 180,E1 10123.387,E2 10123.387} C_VEL
LIN {X 0,Y 397.135,Z 1058.746,A -85,B 0,C 180,E1 10121.274,E2 10121.274} C_VEL
LIN {X 0,Y 406.132,Z 1040.961,A -85,B 0,C 180,E1 10119.07,E2 10119.07} C_VEL
LIN {X 0,Y 416.131,Z 1019.614,A -85,B 0,C 180,E1 10116.858,E2 10116.858} C_VEL
LIN {X 0,Y 423.859,Z 1001.819,A -85,B 0,C 180,E1 10115.294,E2 10115.294} C_VEL
LIN {X 0,Y 431.248,Z 983.435,A -85,B 0,C 180,E1 10113.897,E2 10113.897} C_VEL
LIN {X 0,Y 439.873,Z 959.856,A -85,B 0,C 180,E1 10112.387,E2 10112.387} C_VEL
LIN {X 0,Y 447.084,Z 937.157,A -85,B 0,C 180,E1 10111.192,E2 10111.192} C_VEL
LIN {X 0,Y 452.81,Z 916.851,A -85,B 0,C 180,E1 10110.301,E2 10110.301} C_VEL
LIN {X 0,Y 458.31,Z 894.413,A -85,B 0,C 180,E1 10109.486,E2 10109.486} C_VEL
LIN {X 0,Y 463.494,Z 868.099,A -85,B 0,C 180,E1 10108.737,E2 10108.737} C_VEL
LIN {X 0,Y 466.844,Z 846.239,A -85,B 0,C 180,E1 10108.254,E2 10108.254} C_VEL
LIN {X 0,Y 469.336,Z 823.414,A -85,B 0,C 180,E1 10107.849,E2 10107.849} C_VEL
LIN {X 0,Y 486.575,Z 592.409,A -85,B 0,C 180,E1 10104.307,E2 10104.307} C_VEL
LIN {X 0,Y 490.27,Z 544.258,A -85,B 0,C 180,E1 10103.562,E2 10103.562} C_VEL
LIN {X 0,Y 483.474,Z 531.869,A -85,B 0,C 180,E1 10100.869,E2 10100.869} C_VEL
LIN {X 0,Y 477.568,Z 521.334,A -85,B 0,C 180,E1 10098.115,E2 10098.115} C_VEL
LIN {X 0,Y 472.705,Z 513.071,A -85,B 0,C 180,E1 10095.395,E2 10095.395} C_VEL
LIN {X 0,Y 469.508,Z 507.841,A -85,B 0,C 180,E1 10093.235,E2 10093.235} C_VEL
LIN {X 0,Y 466.964,Z 503.539,A -85,B 0,C 180,E1 10091.111,E2 10091.111} C_VEL
LIN {X 0,Y 464.825,Z 499.782,A -85,B 0,C 180,E1 10088.785,E2 10088.785} C_VEL
LIN {X 0,Y 462.596,Z 495.462,A -85,B 0,C 180,E1 10084.463,E2 10084.463} C_VEL
LIN {X 0,Y 462.505,Z 494.984,A -85,B 0,C 180,E1 10080.248,E2 10080.248} C_VEL
LIN {X 0,Y 464.171,Z 496.363,A -85,B 0,C 180,E1 10076.666,E2 10076.666} C_VEL
LIN {X 0,Y 467.978,Z 501.621,A -85,B 0,C 180,E1 10072.511,E2 10072.511} C_VEL
LIN {X 0,Y 471.522,Z 506.686,A -85,B 0,C 180,E1 10069.863,E2 10069.863} C_VEL
LIN {X 0,Y 475.249,Z 512.134,A -85,B 0,C 180,E1 10067.608,E2 10067.608} C_VEL
LIN {X 0,Y 479.097,Z 517.871,A -85,B 0,C 180,E1 10065.62,E2 10065.62} C_VEL
LIN {X 0,Y 484.537,Z 526.353,A -85,B 0,C 180,E1 10063.177,E2 10063.177} C_VEL
LIN {X 0,Y 491.118,Z 537.054,A -85,B 0,C 180,E1 10060.618,E2 10060.618} C_VEL
LIN {X 0,Y 492.611,Z 539.851,A -85,B 0,C 180,E1 10060.072,E2 10060.072} C_VEL
LIN {X 0,Y 475.348,Z 759.233,A -85,B 0,C 180,E1 10056.595,E2 10056.595} C_VEL
LIN {X 0,Y 469.769,Z 828.979,A -85,B 0,C 180,E1 10055.462,E2 10055.462} C_VEL
LIN {X 0,Y 465.757,Z 858.764,A -85,B 0,C 180,E1 10054.862,E2 10054.862} C_VEL
LIN {X 0,Y 461.576,Z 881.565,A -85,B 0,C 180,E1 10054.264,E2 10054.264} C_VEL
LIN {X 0,Y 456.947,Z 902.75,A -85,B 0,C 180,E1 10053.573,E2 10053.573} C_VEL
LIN {X 0,Y 451.239,Z 925.18,A -85,B 0,C 180,E1 10052.691,E2 10052.691} C_VEL
LIN {X 0,Y 443.501,Z 951.273,A -85,B 0,C 180,E1 10051.431,E2 10051.431} C_VEL
LIN {X 0,Y 436.563,Z 971.919,A -85,B 0,C 180,E1 10050.231,E2 10050.231} C_VEL
LIN {X 0,Y 429.524,Z 991.025,A -85,B 0,C 180,E1 10048.943,E2 10048.943} C_VEL
LIN {X 0,Y 421.511,Z 1011.172,A -85,B 0,C 180,E1 10047.362,E2 10047.362} C_VEL
LIN {X 0,Y 411.141,Z 1035.028,A -85,B 0,C 180,E1 10045.144,E2 10045.144} C_VEL
LIN {X 0,Y 402.828,Z 1052.91,A -85,B 0,C 180,E1 10043.177,E2 10043.177} C_VEL
LIN {X 0,Y 394.824,Z 1069.381,A -85,B 0,C 180,E1 10041.093,E2 10041.093} C_VEL
LIN {X 0,Y 385.859,Z 1087.205,A -85,B 0,C 180,E1 10038.493,E2 10038.493} C_VEL
LIN {X 0,Y 376.453,Z 1105.21,A -85,B 0,C 180,E1 10035.383,E2 10035.383} C_VEL
LIN {X 0,Y 368.965,Z 1119.419,A -85,B 0,C 180,E1 10032.513,E2 10032.513} C_VEL
LIN {X 0,Y 362.391,Z 1131.997,A -85,B 0,C 180,E1 10029.594,E2 10029.594} C_VEL
LIN {X 0,Y 355.301,Z 1146.023,A -85,B 0,C 180,E1 10025.827,E2 10025.827} C_VEL
LIN {X 0,Y 349.077,Z 1158.732,A -85,B 0,C 180,E1 10021.709,E2 10021.709} C_VEL
LIN {X 0,Y 344.933,Z 1167.984,A -85,B 0,C 180,E1 10018.196,E2 10018.196} C_VEL
LIN {X 0,Y 341.777,Z 1175.818,A -85,B 0,C 180,E1 10014.73,E2 10014.73} C_VEL
LIN {X 0,Y 339.146,Z 1183.482,A -85,B 0,C 180,E1 10010.719,E2 10010.719} C_VEL
LIN {X 0,Y 337.212,Z 1190.606,A -85,B 0,C 180,E1 10006.007,E2 10006.007} C_VEL
LIN {X 0,Y 336.376,Z 1195.019,A -85,B 0,C 180,E1 10002.183,E2 10002.183} C_VEL
LIN {X 0,Y 336.059,Z 1198,A -85,B 0,C 180,E1 9998.727,E2 9998.727} C_VEL
LIN {X 0,Y 335.968,Z 1199.998,A -85,B 0,C 180,E1 9995.293,E2 9995.293} C_VEL
LIN {X 0,Y 335.961,Z 1200.996,A -85,B 0,C 180,E1 9992.046,E2 9992.046} C_VEL
LIN {X 0,Y 335.965,Z 1201.114,A -85,B 0,C 180,E1 9988.806,E2 9988.806} C_VEL
LIN {X 0,Y 335.96,Z 1200.282,A -85,B 0,C 180,E1 9985.391,E2 9985.391} C_VEL
LIN {X 0,Y 336.029,Z 1198.473,A -85,B 0,C 180,E1 9981.96,E2 9981.96} C_VEL
LIN {X 0,Y 336.28,Z 1195.682,A -85,B 0,C 180,E1 9978.509,E2 9978.509} C_VEL
LIN {X 0,Y 336.927,Z 1191.898,A -85,B 0,C 180,E1 9975.037,E2 9975.037} C_VEL
LIN {X 0,Y 338.06,Z 1187.095,A -85,B 0,C 180,E1 9971.55,E2 9971.55} C_VEL
LIN {X 0,Y 339.93,Z 1180.971,A -85,B 0,C 180,E1 9967.905,E2 9967.905} C_VEL
LIN {X 0,Y 342.95,Z 1172.85,A -85,B 0,C 180,E1 9963.88,E2 9963.88} C_VEL
LIN {X 0,Y 347.659,Z 1161.798,A -85,B 0,C 180,E1 9959.399,E2 9959.399} C_VEL
LIN {X 0,Y 352.576,Z 1151.35,A -85,B 0,C 180,E1 9955.839,E2 9955.839} C_VEL
LIN {X 0,Y 358.205,Z 1140.063,A -85,B 0,C 180,E1 9952.517,E2 9952.517} C_VEL
LIN {X 0,Y 365.903,Z 1125.388,A -85,B 0,C 180,E1 9948.809,E2 9948.809} C_VEL
LIN {X 0,Y 374.369,Z 1109.095,A -85,B 0,C 180,E1 9945.377,E2 9945.377} C_VEL
LIN {X 0,Y 381.689,Z 1095.058,A -85,B 0,C 180,E1 9942.82,E2 9942.82} C_VEL
LIN {X 0,Y 389.669,Z 1079.524,A -85,B 0,C 180,E1 9940.351,E2 9940.351} C_VEL
LIN {X 0,Y 399.864,Z 1059.021,A -85,B 0,C 180,E1 9937.564,E2 9937.564} C_VEL
LIN {X 0,Y 408.928,Z 1039.66,A -85,B 0,C 180,E1 9935.351,E2 9935.351} C_VEL
LIN {X 0,Y 416.878,Z 1021.815,A -85,B 0,C 180,E1 9933.591,E2 9933.591} C_VEL
LIN {X 0,Y 425.167,Z 1002.011,A -85,B 0,C 180,E1 9931.899,E2 9931.899} C_VEL
LIN {X 0,Y 434.748,Z 976.806,A -85,B 0,C 180,E1 9930.092,E2 9930.092} C_VEL
LIN {X 0,Y 441.451,Z 957.223,A -85,B 0,C 180,E1 9928.905,E2 9928.905} C_VEL
LIN {X 0,Y 447.468,Z 937.896,A -85,B 0,C 180,E1 9927.901,E2 9927.901} C_VEL
LIN {X 0,Y 453.278,Z 917.038,A -85,B 0,C 180,E1 9926.978,E2 9926.978} C_VEL
LIN {X 0,Y 459.591,Z 890.909,A -85,B 0,C 180,E1 9926.027,E2 9926.027} C_VEL
LIN {X 0,Y 464.488,Z 865.429,A -85,B 0,C 180,E1 9925.306,E2 9925.306} C_VEL
LIN {X 0,Y 467.91,Z 843.347,A -85,B 0,C 180,E1 9924.817,E2 9924.817} C_VEL
LIN {X 0,Y 470.607,Z 818.944,A -85,B 0,C 180,E1 9924.373,E2 9924.373} C_VEL
LIN {X 0,Y 487.926,Z 596.733,A -85,B 0,C 180,E1 9920.832,E2 9920.832} C_VEL
LIN {X 0,Y 492.454,Z 539.458,A -85,B 0,C 180,E1 9919.917,E2 9919.917} C_VEL
LIN {X 0,Y 485.145,Z 527.366,A -85,B 0,C 180,E1 9917.141,E2 9917.141} C_VEL
LIN {X 0,Y 479.167,Z 518.069,A -85,B 0,C 180,E1 9914.502,E2 9914.502} C_VEL
LIN {X 0,Y 475.071,Z 511.962,A -85,B 0,C 180,E1 9912.397,E2 9912.397} C_VEL
LIN {X 0,Y 470.631,Z 505.373,A -85,B 0,C 180,E1 9909.662,E2 9909.662} C_VEL
LIN {X 0,Y 467.212,Z 500.658,A -85,B 0,C 180,E1 9907.007,E2 9907.007} C_VEL
LIN {X 0,Y 463.694,Z 495.834,A -85,B 0,C 180,E1 9902.967,E2 9902.967} C_VEL
LIN {X 0,Y 462.033,Z 494.684,A -85,B 0,C 180,E1 9898.636,E2 9898.636} C_VEL
LIN {X 0,Y 462.532,Z 495.581,A -85,B 0,C 180,E1 9894.791,E2 9894.791} C_VEL
LIN {X 0,Y 465.235,Z 500.605,A -85,B 0,C 180,E1 9890.349,E2 9890.349} C_VEL
LIN {X 0,Y 467.966,Z 505.405,A -85,B 0,C 180,E1 9887.725,E2 9887.725} C_VEL
LIN {X 0,Y 470.799,Z 510.135,A -85,B 0,C 180,E1 9885.612,E2 9885.612} C_VEL
LIN {X 0,Y 475.011,Z 517.156,A -85,B 0,C 180,E1 9883.05,E2 9883.05} C_VEL
LIN {X 0,Y 479.972,Z 525.78,A -85,B 0,C 180,E1 9880.53,E2 9880.53} C_VEL
LIN {X 0,Y 485.808,Z 536.241,A -85,B 0,C 180,E1 9878.001,E2 9878.001} C_VEL
LIN {X 0,Y 490.148,Z 544.369,A -85,B 0,C 180,E1 9876.328,E2 9876.328} C_VEL
LIN {X 0,Y 473.529,Z 764.932,A -85,B 0,C 180,E1 9872.959,E2 9872.959} C_VEL
LIN {X 0,Y 468.377,Z 832.311,A -85,B 0,C 180,E1 9871.905,E2 9871.905} C_VEL
LIN {X 0,Y 464.572,Z 860.876,A -85,B 0,C 180,E1 9871.337,E2 9871.337} C_VEL
LIN {X 0,Y 460.538,Z 882.882,A -85,B 0,C 180,E1 9870.773,E2 9870.773} C_VEL
LIN {X 0,Y 455.585,Z 905.405,A -85,B 0,C 180,E1 9870.039,E2 9870.039} C_VEL
LIN {X 0,Y 448.652,Z 931.527,A -85,B 0,C 180,E1 9868.971,E2 9868.971} C_VEL
LIN {X 0,Y 442.153,Z 952.537,A -85,B 0,C 180,E1 9867.916,E2 9867.916} C_VEL
LIN {X 0,Y 435.583,Z 971.552,A -85,B 0,C 180,E1 9866.794,E2 9866.794} C_VEL
LIN {X 0,Y 427.136,Z 993.785,A -85,B 0,C 180,E1 9865.251,E2 9865.251} C_VEL
LIN {X 0,Y 418.087,Z 1014.963,A -85,B 0,C 180,E1 9863.472,E2 9863.472} C_VEL
LIN {X 0,Y 410.011,Z 1032.564,A -85,B 0,C 180,E1 9861.744,E2 9861.744} C_VEL
LIN {X 0,Y 400.716,Z 1051.686,A -85,B 0,C 180,E1 9859.551,E2 9859.551} C_VEL
LIN {X 0,Y 391.012,Z 1070.242,A -85,B 0,C 180,E1 9857,E2 9857} C_VEL
LIN {X 0,Y 382.96,Z 1085.044,A -85,B 0,C 180,E1 9854.615,E2 9854.615} C_VEL
LIN {X 0,Y 374.944,Z 1099.437,A -85,B 0,C 180,E1 9851.924,E2 9851.924} C_VEL
LIN {X 0,Y 365.726,Z 1115.62,A -85,B 0,C 180,E1 9848.311,E2 9848.311} C_VEL
LIN {X 0,Y 359.082,Z 1127.307,A -85,B 0,C 180,E1 9845.198,E2 9845.198} C_VEL
LIN {X 0,Y 353.037,Z 1138.244,A -85,B 0,C 180,E1 9841.789,E2 9841.789} C_VEL
LIN {X 0,Y 346.9,Z 1149.843,A -85,B 0,C 180,E1 9837.406,E2 9837.406} C_VEL
LIN {X 0,Y 343.02,Z 1157.839,A -85,B 0,C 180,E1 9833.72,E2 9833.72} C_VEL
LIN {X 0,Y 340.009,Z 1164.942,A -85,B 0,C 180,E1 9829.767,E2 9829.767} C_VEL
LIN {X 0,Y 337.727,Z 1171.435,A -85,B 0,C 180,E1 9825.102,E2 9825.102} C_VEL
LIN {X 0,Y 336.718,Z 1175.224,A -85,B 0,C 180,E1 9821.476,E2 9821.476} C_VEL
LIN {X 0,Y 336.238,Z 1177.882,A -85,B 0,C 180,E1 9818,E2 9818} C_VEL
LIN {X 0,Y 336.034,Z 1179.58,A -85,B 0,C 180,E1 9814.572,E2 9814.572} C_VEL
LIN {X 0,Y 335.993,Z 1180.358,A -85,B 0,C 180,E1 9811.194,E2 9811.194} C_VEL
LIN {X 0,Y 336.001,Z 1180.221,A -85,B 0,C 180,E1 9807.613,E2 9807.613} C_VEL
LIN {X 0,Y 336.134,Z 1178.792,A -85,B 0,C 180,E1 9803.338,E2 9803.338} C_VEL
LIN {X 0,Y 336.572,Z 1175.926,A -85,B 0,C 180,E1 9799.213,E2 9799.213} C_VEL
LIN {X 0,Y 337.462,Z 1172.343,A -85,B 0,C 180,E1 9795.589,E2 9795.589} C_VEL
LIN {X 0,Y 338.971,Z 1167.686,A -85,B 0,C 180,E1 9791.958,E2 9791.958} C_VEL
LIN {X 0,Y 341.869,Z 1160.575,A -85,B 0,C 180,E1 9787.553,E2 9787.553} C_VEL
LIN {X 0,Y 345.877,Z 1151.908,A -85,B 0,C 180,E1 9783.38,E2 9783.38} C_VEL
LIN {X 0,Y 350.419,Z 1143.099,A -85,B 0,C 180,E1 9779.836,E2 9779.836} C_VEL
LIN {X 0,Y 356.837,Z 1131.518,A -85,B 0,C 180,E1 9775.916,E2 9775.916} C_VEL
LIN {X 0,Y 364.24,Z 1118.286,A -85,B 0,C 180,E1 9772.255,E2 9772.255} C_VEL
LIN {X 0,Y 364.364,Z 1118.068,A -85,B 0,C 180,E1 9772.2,E2 9772.2} C_VEL
LIN {X 0,Y 365.75,Z 1114.343,A -85,B 0,C 180,E1 9771.153,E2 9771.153} C_VEL
LIN {X 0,Y 366.708,Z 1104.613,A -85,B 0,C 180,E1 9768.201,E2 9768.201} C_VEL
LIN {X 0,Y 368.215,Z 1100.984,A -85,B 0,C 180,E1 9767.364,E2 9767.364} C_VEL
LIN {X 0,Y 377.172,Z 1085.44,A -85,B 0,C 180,E1 9764.417,E2 9764.417} C_VEL
LIN {X 0,Y 385.777,Z 1070.14,A -85,B 0,C 180,E1 9761.939,E2 9761.939} C_VEL
LIN {X 0,Y 396.361,Z 1050.404,A -85,B 0,C 180,E1 9759.245,E2 9759.245} C_VEL
LIN {X 0,Y 405.494,Z 1032.159,A -85,B 0,C 180,E1 9757.167,E2 9757.167} C_VEL
LIN {X 0,Y 413.774,Z 1014.567,A -85,B 0,C 180,E1 9755.448,E2 9755.448} C_VEL
LIN {X 0,Y 423.618,Z 991.869,A -85,B 0,C 180,E1 9753.572,E2 9753.572} C_VEL
LIN {X 0,Y 431.697,Z 971.069,A -85,B 0,C 180,E1 9752.148,E2 9752.148} C_VEL
LIN {X 0,Y 438.323,Z 952.314,A -85,B 0,C 180,E1 9751.054,E2 9751.054} C_VEL
LIN {X 0,Y 444.707,Z 932.124,A -85,B 0,C 180,E1 9750.046,E2 9750.046} C_VEL
LIN {X 0,Y 451.932,Z 905.585,A -85,B 0,C 180,E1 9748.966,E2 9748.966} C_VEL
LIN {X 0,Y 456.967,Z 883.192,A -85,B 0,C 180,E1 9748.241,E2 9748.241} C_VEL
LIN {X 0,Y 461.089,Z 861.186,A -85,B 0,C 180,E1 9747.679,E2 9747.679} C_VEL
LIN {X 0,Y 464.921,Z 833.485,A -85,B 0,C 180,E1 9747.129,E2 9747.129} C_VEL
LIN {X 0,Y 469.141,Z 780.653,A -85,B 0,C 180,E1 9746.299,E2 9746.299} C_VEL
LIN {X 0,Y 486.364,Z 557.43,A -85,B 0,C 180,E1 9742.894,E2 9742.894} C_VEL
LIN {X 0,Y 486.955,Z 549.159,A -85,B 0,C 180,E1 9742.746,E2 9742.746} C_VEL
LIN {X 0,Y 481.348,Z 538.681,A -85,B 0,C 180,E1 9740.425,E2 9740.425} C_VEL
LIN {X 0,Y 475.78,Z 528.541,A -85,B 0,C 180,E1 9737.742,E2 9737.742} C_VEL
LIN {X 0,Y 471.174,Z 520.525,A -85,B 0,C 180,E1 9735.083,E2 9735.083} C_VEL
LIN {X 0,Y 468.13,Z 515.42,A -85,B 0,C 180,E1 9732.96,E2 9732.96} C_VEL
LIN {X 0,Y 465.731,Z 511.247,A -85,B 0,C 180,E1 9730.89,E2 9730.89} C_VEL
LIN {X 0,Y 463.759,Z 507.665,A -85,B 0,C 180,E1 9728.681,E2 9728.681} C_VEL
LIN {X 0,Y 461.589,Z 503.37,A -85,B 0,C 180,E1 9724.348,E2 9724.348} C_VEL
LIN {X 0,Y 461.53,Z 502.926,A -85,B 0,C 180,E1 9720.248,E2 9720.248} C_VEL
LIN {X 0,Y 463.107,Z 504.239,A -85,B 0,C 180,E1 9716.782,E2 9716.782} C_VEL
LIN {X 0,Y 466.837,Z 509.544,A -85,B 0,C 180,E1 9712.616,E2 9712.616} C_VEL
LIN {X 0,Y 470.16,Z 514.369,A -85,B 0,C 180,E1 9710.081,E2 9710.081} C_VEL
LIN {X 0,Y 473.819,Z 519.826,A -85,B 0,C 180,E1 9707.817,E2 9707.817} C_VEL
LIN {X 0,Y 478.329,Z 526.599,A -85,B 0,C 180,E1 9705.472,E2 9705.472} C_VEL
LIN {X 0,Y 484.183,Z 536.155,A -85,B 0,C 180,E1 9702.855,E2 9702.855} C_VEL
LIN {X 0,Y 489.251,Z 544.752,A -85,B 0,C 180,E1 9700.867,E2 9700.867} C_VEL
LIN {X 0,Y 471.474,Z 765.493,A -85,B 0,C 180,E1 9697.376,E2 9697.376} C_VEL
LIN {X 0,Y 466.212,Z 829.42,A -85,B 0,C 180,E1 9696.338,E2 9696.338} C_VEL
LIN {X 0,Y 462.086,Z 859.249,A -85,B 0,C 180,E1 9695.738,E2 9695.738} C_VEL
LIN {X 0,Y 457.867,Z 881.769,A -85,B 0,C 180,E1 9695.151,E2 9695.151} C_VEL
LIN {X 0,Y 453.188,Z 902.739,A -85,B 0,C 180,E1 9694.473,E2 9694.473} C_VEL
LIN {X 0,Y 447.288,Z 925.443,A -85,B 0,C 180,E1 9693.586,E2 9693.586} C_VEL
LIN {X 0,Y 439.248,Z 951.864,A -85,B 0,C 180,E1 9692.312,E2 9692.312} C_VEL
LIN {X 0,Y 432.162,Z 972.412,A -85,B 0,C 180,E1 9691.12,E2 9691.12} C_VEL
LIN {X 0,Y 424.663,Z 992.224,A -85,B 0,C 180,E1 9689.78,E2 9689.78} C_VEL
LIN {X 0,Y 415.227,Z 1015.208,A -85,B 0,C 180,E1 9687.954,E2 9687.954} C_VEL
LIN {X 0,Y 405.288,Z 1037.04,A -85,B 0,C 180,E1 9685.863,E2 9685.863} C_VEL
LIN {X 0,Y 397.021,Z 1054.252,A -85,B 0,C 180,E1 9683.941,E2 9683.941} C_VEL
LIN {X 0,Y 388.402,Z 1071.4,A -85,B 0,C 180,E1 9681.736,E2 9681.736} C_VEL
LIN {X 0,Y 377.413,Z 1092.224,A -85,B 0,C 180,E1 9678.568,E2 9678.568} C_VEL
LIN {X 0,Y 369.25,Z 1107.274,A -85,B 0,C 180,E1 9675.855,E2 9675.855} C_VEL
LIN {X 0,Y 361.841,Z 1120.824,A -85,B 0,C 180,E1 9673.042,E2 9673.042} C_VEL
LIN {X 0,Y 353.536,Z 1136.262,A -85,B 0,C 180,E1 9669.31,E2 9669.31} C_VEL
LIN {X 0,Y 346.438,Z 1149.5,A -85,B 0,C 180,E1 9665.458,E2 9665.458} C_VEL
LIN {X 0,Y 341.347,Z 1159.645,A -85,B 0,C 180,E1 9662.018,E2 9662.018} C_VEL
LIN {X 0,Y 337.18,Z 1168.551,A -85,B 0,C 180,E1 9658.517,E2 9658.517} C_VEL
LIN {X 0,Y 333.239,Z 1178.123,A -85,B 0,C 180,E1 9654.083,E2 9654.083} C_VEL
LIN {X 0,Y 330.552,Z 1185.781,A -85,B 0,C 180,E1 9649.618,E2 9649.618} C_VEL
LIN {X 0,Y 329.16,Z 1191,A -85,B 0,C 180,E1 9645.866,E2 9645.866} C_VEL
LIN {X 0,Y 328.375,Z 1195.039,A -85,B 0,C 180,E1 9642.193,E2 9642.193} C_VEL
LIN {X 0,Y 328.061,Z 1197.869,A -85,B 0,C 180,E1 9638.765,E2 9638.765} C_VEL
LIN {X 0,Y 327.97,Z 1199.749,A -85,B 0,C 180,E1 9635.423,E2 9635.423} C_VEL
LIN {X 0,Y 327.964,Z 1200.748,A -85,B 0,C 180,E1 9632.096,E2 9632.096} C_VEL
LIN {X 0,Y 327.969,Z 1200.867,A -85,B 0,C 180,E1 9628.777,E2 9628.777} C_VEL
LIN {X 0,Y 327.962,Z 1200.105,A -85,B 0,C 180,E1 9625.453,E2 9625.453} C_VEL
LIN {X 0,Y 328.031,Z 1198.342,A -85,B 0,C 180,E1 9621.939,E2 9621.939} C_VEL
LIN {X 0,Y 328.291,Z 1195.596,A -85,B 0,C 180,E1 9618.403,E2 9618.403} C_VEL
LIN {X 0,Y 328.969,Z 1191.856,A -85,B 0,C 180,E1 9614.847,E2 9614.847} C_VEL
LIN {X 0,Y 330.231,Z 1186.832,A -85,B 0,C 180,E1 9611.096,E2 9611.096} C_VEL
LIN {X 0,Y 332.135,Z 1180.981,A -85,B 0,C 180,E1 9607.522,E2 9607.522} C_VEL
LIN {X 0,Y 335.236,Z 1173.061,A -85,B 0,C 180,E1 9603.482,E2 9603.482} C_VEL
LIN {X 0,Y 340.443,Z 1161.517,A -85,B 0,C 180,E1 9598.678,E2 9598.678} C_VEL
LIN {X 0,Y 345.609,Z 1151.063,A -85,B 0,C 180,E1 9595.052,E2 9595.052} C_VEL
LIN {X 0,Y 351.383,Z 1140.047,A -85,B 0,C 180,E1 9591.756,E2 9591.756} C_VEL
LIN {X 0,Y 359.568,Z 1125.084,A -85,B 0,C 180,E1 9587.92,E2 9587.92} C_VEL
LIN {X 0,Y 368.399,Z 1108.758,A -85,B 0,C 180,E1 9584.448,E2 9584.448} C_VEL
LIN {X 0,Y 375.988,Z 1094.734,A -85,B 0,C 180,E1 9581.874,E2 9581.874} C_VEL
LIN {X 0,Y 384.514,Z 1078.717,A -85,B 0,C 180,E1 9579.32,E2 9579.32} C_VEL
LIN {X 0,Y 395.62,Z 1056.955,A -85,B 0,C 180,E1 9576.393,E2 9576.393} C_VEL
LIN {X 0,Y 404.103,Z 1039.366,A -85,B 0,C 180,E1 9574.392,E2 9574.392} C_VEL
LIN {X 0,Y 412.133,Z 1021.828,A -85,B 0,C 180,E1 9572.663,E2 9572.663} C_VEL
LIN {X 0,Y 420.832,Z 1001.584,A -85,B 0,C 180,E1 9570.938,E2 9570.938} C_VEL
LIN {X 0,Y 430.527,Z 976.67,A -85,B 0,C 180,E1 9569.162,E2 9569.162} C_VEL
LIN {X 0,Y 437.56,Z 956.578,A -85,B 0,C 180,E1 9567.955,E2 9567.955} C_VEL
LIN {X 0,Y 444.031,Z 936.151,A -85,B 0,C 180,E1 9566.909,E2 9566.909} C_VEL
LIN {X 0,Y 451.046,Z 911.168,A -85,B 0,C 180,E1 9565.839,E2 9565.839} C_VEL
LIN {X 0,Y 457.11,Z 884.851,A -85,B 0,C 180,E1 9564.949,E2 9564.949} C_VEL
LIN {X 0,Y 461.271,Z 863.136,A -85,B 0,C 180,E1 9564.362,E2 9564.362} C_VEL
LIN {X 0,Y 464.788,Z 840.26,A -85,B 0,C 180,E1 9563.871,E2 9563.871} C_VEL
LIN {X 0,Y 468.189,Z 805.896,A -85,B 0,C 180,E1 9563.276,E2 9563.276} C_VEL
LIN {X 0,Y 486.233,Z 579.829,A -85,B 0,C 180,E1 9559.692,E2 9559.692} C_VEL
